Omron CX-Programmer project NewProject (CX-Programmer 9.80)

# PLC IN650_850: CJ2M CPU12
I/O table (CPU CJ2M-CPU12): rack 0 slot 1 CJ1W-ID211; rack 0 slot 2 CJ1W-ID211; rack 0 slot 3 CJ1W-OD212; rack 0 slot 4 CJ1W-OD212; rack 0 slot 5 CJ1W-OD212

## Global symbols (name address type ; comment)
ACC_Target_Frequency H31 DINT
ACC_accel_decel H30 UINT
AC_Drive_Fault W151.12 BOOL
AC_Drive_OK 1.07 BOOL  ; Drive OK output from infeed conveyor
ADV_ACC D882 DINT
ADV_ACC_4ms D1100 UINT
ADV_DEC D884 DINT
ADV_DEC_4ms D1104 UINT
ADV_Movement_Calcs Vel_ACC_DEC_Scale
ADV_Vel D886 DINT
Air_Pressure_Check T0160 TIMER  ; Debounce delay for Air Pressure
Air_Pressure_Fault W151.02 BOOL  ; Air Pressure Fault
Air_Pressure_OK 0.04 BOOL  ; Air Pressure switch
Analog_IO_Type D20001 CHANNEL  ; Analog input and output types.  Bit pattern of 1010101000000001 (#AA01) means all inputs are 4-20 mA and the output are 0 - 10VDC).
Analog_IO_Use_Config D20000 CHANNEL  ; #71 means that Inputs 1, 2 and 3 are used (bits 4, 5 and 6 on makes up 7 HEX) and output 1 is used (bit 0 on makes up 1 HEX).
2008 CHANNEL  ; top Vac sensor
D10000 CHANNEL  ; Vacuum graph 1 starting word
D10001 CHANNEL  ; top Vac scaled output
D10022 CHANNEL  ; scaled_measured_height_forHMI
D2041 CHANNEL  ; Unscaled Point A in slope
D2042 CHANNEL  ; Scaled Point B in slope
D2043 CHANNEL  ; Unscaled Point B in slope
D920 CHANNEL  ; Present value 1
D921 CHANNEL  ; Loop 2 Present value
D922 CHANNEL  ; Loop 3 Present value
D925 CHANNEL  ; Setpoint 1
T0226 BOOL  ; Delay down for lowering
T1103 BOOL  ; idel film time out
W497.00 BOOL  ; Temp bit HMI
Average_tray_height D2036 UINT  ; Average height of trays
Average_trays Average
Beginning_of_Cycle W202.06 BOOL  ; Beginning of the cycle
Break_Recover_Timer T1102 TIMER  ; Printer Film Break Delay
Calc_TPM TPM_Calc
Clear_Film_parameter_changed D2204.02 BOOL  ; Clear film parameter has changed
Close_Tool_Latch W200.12 BOOL
Cool_Timer T0124 TIMER  ; Cool Timer
CtoF C_to_F
Current1 D3005 CHANNEL  ; Stroom solid state 1
Current2 D3006 CHANNEL  ; Stroom solid state 2
Current3 D3007 CHANNEL  ; Stroom solid state 3
Current4 D3008 CHANNEL  ; Stroom solid state 4
Dancing_Timer T0203 TIMER  ; Dancing Timer
Dancing_Tray_Stop_Bit W200.14 BOOL
Data_Recipe_0 E0 CHANNEL[250]  ; All of the data for Recipe 0
Data_Recipe_1 E250 CHANNEL[250]  ; All of the data for Recipe 1
Data_Recipe_10 E2500 CHANNEL[250]  ; All of the data for Recipe 10
Data_Recipe_11 E2750 CHANNEL[250]  ; All of the data for Recipe 11
Data_Recipe_12 E3000 CHANNEL[250]  ; All of the data for Recipe 12
Data_Recipe_13 E3250 CHANNEL[250]  ; All of the data for Recipe 13
Data_Recipe_14 E3500 CHANNEL[250]  ; All of the data for Recipe 14
Data_Recipe_15 E3750 CHANNEL[250]  ; All of the data for Recipe 15
Data_Recipe_16 E4000 CHANNEL[250]  ; All of the data for Recipe 16
Data_Recipe_17 E4250 CHANNEL[250]  ; All of the data for Recipe 17
Data_Recipe_18 E4500 CHANNEL[250]  ; All of the data for Recipe 18
Data_Recipe_19 E4750 CHANNEL[250]  ; All of the data for Recipe 19
Data_Recipe_2 E500 CHANNEL[250]  ; All of the data for Recipe 2
Data_Recipe_20 E5000 CHANNEL[250]  ; All of the data for Recipe 20
Data_Recipe_21 E5250 CHANNEL[250]  ; All of the data for Recipe 21
Data_Recipe_22 E5500 CHANNEL[250]  ; All of the data for Recipe 22
Data_Recipe_23 E5750 CHANNEL[250]  ; All of the data for Recipe 23
Data_Recipe_24 E6000 CHANNEL[250]  ; All of the data for Recipe 24
Data_Recipe_25 E6250 CHANNEL[250]  ; All of the data for Recipe 25
Data_Recipe_26 E6500 CHANNEL[250]  ; All of the data for Recipe 26
Data_Recipe_27 E6750 CHANNEL[250]  ; All of the data for Recipe 27
Data_Recipe_28 E7000 CHANNEL[250]  ; All of the data for Recipe 28
Data_Recipe_29 E7250 CHANNEL[250]  ; All of the data for Recipe 29
Data_Recipe_3 E750 CHANNEL[250]  ; All of the data for Recipe 3
Data_Recipe_30 E7500 CHANNEL[250]  ; All of the data for Recipe 30
Data_Recipe_31 E7750 CHANNEL[250]  ; All of the data for Recipe 31
Data_Recipe_32 E8000 CHANNEL[250]  ; All of the data for Recipe 32
Data_Recipe_33 E8250 CHANNEL[250]  ; All of the data for Recipe 33
Data_Recipe_34 E8500 CHANNEL[250]  ; All of the data for Recipe 34
Data_Recipe_35 E8750 CHANNEL[250]  ; All of the data for Recipe 35
Data_Recipe_36 E9000 CHANNEL[250]  ; All of the data for Recipe 36
Data_Recipe_37 E9250 CHANNEL[250]  ; All of the data for Recipe 37
Data_Recipe_38 E9500 CHANNEL[250]  ; All of the data for Recipe 38
Data_Recipe_39 E9750 CHANNEL[250]  ; All of the data for Recipe 39
Data_Recipe_4 E1000 CHANNEL[250]  ; All of the data for Recipe 4
Data_Recipe_40 E10000 CHANNEL[250]  ; All of the data for Recipe 40
Data_Recipe_41 E10250 CHANNEL[250]  ; All of the data for Recipe 41
Data_Recipe_42 E10500 CHANNEL[250]  ; All of the data for Recipe 42
Data_Recipe_43 E10750 CHANNEL[250]  ; All of the data for Recipe 43
Data_Recipe_44 E11000 CHANNEL[250]  ; All of the data for Recipe 44
Data_Recipe_45 E11250 CHANNEL[250]  ; All of the data for Recipe 45
Data_Recipe_46 E11500 CHANNEL[250]  ; All of the data for Recipe 46
Data_Recipe_47 E11750 CHANNEL[250]  ; All of the data for Recipe 47
Data_Recipe_48 E12000 CHANNEL[250]  ; All of the data for Recipe 48
Data_Recipe_49 E12250 CHANNEL[250]  ; All of the data for Recipe 49
Data_Recipe_5 E1250 CHANNEL[250]  ; All of the data for Recipe 5
Data_Recipe_50 E12500 CHANNEL[250]  ; All of the data for Recipe 50
Data_Recipe_51 E12750 CHANNEL[250]  ; All of the data for Recipe 51
Data_Recipe_52 E13000 CHANNEL[250]  ; All of the data for Recipe 52
Data_Recipe_53 E13250 CHANNEL[250]  ; All of the data for Recipe 53
Data_Recipe_54 E13500 CHANNEL[250]  ; All of the data for Recipe 54
Data_Recipe_55 E13750 CHANNEL[250]  ; All of the data for Recipe 55
Data_Recipe_56 E14000 CHANNEL[250]  ; All of the data for Recipe 56
Data_Recipe_57 E14250 CHANNEL[250]  ; All of the data for Recipe 57
Data_Recipe_58 E14500 CHANNEL[250]  ; All of the data for Recipe 58
Data_Recipe_59 E14750 CHANNEL[250]  ; All of the data for Recipe 59
Data_Recipe_6 E1500 CHANNEL[250]  ; All of the data for Recipe 6
Data_Recipe_60 E15000 CHANNEL[250]  ; All of the data for Recipe 60
Data_Recipe_61 E15250 CHANNEL[250]  ; All of the data for Recipe 61
Data_Recipe_62 E15500 CHANNEL[250]  ; All of the data for Recipe 62
Data_Recipe_63 E15750 CHANNEL[250]  ; All of the data for Recipe 63
Data_Recipe_64 E16000 CHANNEL[250]  ; All of the data for Recipe 64
Data_Recipe_65 E16250 CHANNEL[250]  ; All of the data for Recipe 65
Data_Recipe_66 E16500 CHANNEL[250]  ; All of the data for Recipe 66
Data_Recipe_67 E16750 CHANNEL[250]  ; All of the data for Recipe 67
Data_Recipe_68 E17000 CHANNEL[250]  ; All of the data for Recipe 68
Data_Recipe_69 E17250 CHANNEL[250]  ; All of the data for Recipe 69
Data_Recipe_7 E1750 CHANNEL[250]  ; All of the data for Recipe 7
Data_Recipe_70 E17500 CHANNEL[250]  ; All of the data for Recipe 70
Data_Recipe_71 E17750 CHANNEL[250]  ; All of the data for Recipe 71
Data_Recipe_72 E18000 CHANNEL[250]  ; All of the data for Recipe 72
Data_Recipe_73 E18250 CHANNEL[250]  ; All of the data for Recipe 73
Data_Recipe_74 E18500 CHANNEL[250]  ; All of the data for Recipe 74
Data_Recipe_75 E18750 CHANNEL[250]  ; All of the data for Recipe 75
Data_Recipe_76 E19000 CHANNEL[250]  ; All of the data for Recipe 76
Data_Recipe_77 E19250 CHANNEL[250]  ; All of the data for Recipe 77
Data_Recipe_78 E19500 CHANNEL[250]  ; All of the data for Recipe 78
Data_Recipe_79 E19750 CHANNEL[250]  ; All of the data for Recipe 79
Data_Recipe_8 E2000 CHANNEL[250]  ; All of the data for Recipe 8
Data_Recipe_80 E20000 CHANNEL[250]  ; All of the data for Recipe 80
Data_Recipe_81 E20250 CHANNEL[250]  ; All of the data for Recipe 81
Data_Recipe_82 E20500 CHANNEL[250]  ; All of the data for Recipe 82
Data_Recipe_83 E20750 CHANNEL[250]  ; All of the data for Recipe 83
Data_Recipe_84 E21000 CHANNEL[250]  ; All of the data for Recipe 84
Data_Recipe_85 E21250 CHANNEL[250]  ; All of the data for Recipe 85
Data_Recipe_86 E21500 CHANNEL[250]  ; All of the data for Recipe 86
Data_Recipe_87 E21750 CHANNEL[250]  ; All of the data for Recipe 87
Data_Recipe_88 E22000 CHANNEL[250]  ; All of the data for Recipe 88
Data_Recipe_89 E22250 CHANNEL[250]  ; All of the data for Recipe 89
Data_Recipe_9 E2250 CHANNEL[250]  ; All of the data for Recipe 9
Data_Recipe_90 E22500 CHANNEL[250]  ; All of the data for Recipe 90
Data_Recipe_91 E22750 CHANNEL[250]  ; All of the data for Recipe 91
Data_Recipe_92 E23000 CHANNEL[250]  ; All of the data for Recipe 92
Data_Recipe_93 E23250 CHANNEL[250]  ; All of the data for Recipe 93
Data_Recipe_94 E23500 CHANNEL[250]  ; All of the data for Recipe 94
Data_Recipe_95 E23750 CHANNEL[250]  ; All of the data for Recipe 95
Data_Recipe_96 E24000 CHANNEL[250]  ; All of the data for Recipe 96
Data_Recipe_97 E24250 CHANNEL[250]  ; All of the data for Recipe 97
Data_Recipe_98 E24500 CHANNEL[250]  ; All of the data for Recipe 98
Data_Recipe_99 E24750 CHANNEL[250]  ; All of the data for Recipe 99
Debounce_TS1 T0100 TIMER  ; Debounce timer for sensor at Tray Stop 1
Debounce_TS2 T0101 TIMER  ; Debounce timer for sensor at Tray Stop 2
Debounce_TS3 T0102 TIMER  ; Debounce timer for sensor at Tray Stop 3
Debounce_TS4 T0103 TIMER  ; Debounce timer for sensor at Tray Stop 4
Debounce_TS5 T0104 TIMER  ; Debounce timer for sensor at Tray Stop 5
Default_Recipe_Data E26000 CHANNEL[250]  ; Default recipe data used when erasing a recipe
Delay_on_upstream D280 UINT
Demo_Mode W200.10 BOOL  ; With or without trays
Demo_Mode_No_Trays W201.00 BOOL
Demo_Mode_With_Trays W201.01 BOOL
Disable_Gas_Delay W250.05 BOOL  ; Disables Input on the HMI
Disable_Gas_Duration W250.06 BOOL  ; Disables Input on the HMI
Disable_Gas_Pressure W250.07 BOOL  ; Disables Input on the HMI
Disable_Seal_Delay W250.10 BOOL  ; Disables Input on the HMI
Disable_Seal_Duration W250.11 BOOL  ; Disables Input on the HMI
Disable_Stepper_out 2961.04 BOOL
Disable_Tool_Open_Delay W250.12 BOOL  ; Disables Input on the HMI
Disable_Vac_Bottom_Delay W250.01 BOOL  ; Disables Input on the HMI
Disable_Vac_Extra W250.04 BOOL  ; Disables Input on the HMI
Disable_Vac_Top_Delay W250.00 BOOL  ; Disables Input on the HMI
Disable_Vac_duration W250.02 BOOL  ; Disables Input on the HMI
Disable_Vac_pressure W250.03 BOOL  ; Disables Input on the HMI
Disable_Vent_Pressure W250.09 BOOL  ; Disables Input on the HMI
Disable_Vent_Top_Delay W250.08 BOOL  ; Disables Input on the HMI
Disable_by_Pressure W202.08 BOOL  ; Disable vac, gas and vent by pressure buttons
Door_Open_Fault W151.01 BOOL  ; Door open
DownStream_Alarm W154.00 BOOL  ; Downstream alarm message bit
Downstream_bypass D2009.13 BOOL  ; Bypass Downstream input
Enable_Analog_Out 2000.00 BOOL  ; enables analog output for speed reference to AC Drive.
Execute_slow_down D2204.01 BOOL
Eye_mark_selection D2300.00 BOOL  ; Single Eye Mark per move selected
FILMREG_ESTOP_DECEL H50 UINT  ; H50 Film Reg E-Stop Decel
FILMREG_ESTOP_FREQ H51 DINT  ; H51/H52 Film Reg E-Stop Target Freq
FILM_DIST_REVYANK_REGIST D1158 DINT
Fault_Exists W156.15 BOOL  ; A fault exists
File_Mem_Operation_Flag A343.13 BOOL  ; File memory operation in progress.
File_Write_Read_Destination D1450 WORD[4]  ; Destination word for FWRIT and FREAD instructions
FilmReg_Started W203.15 BOOL  ; Film Feed with Registration Started
FilmScaling Film_Scaling
Film_Accel_Rate H0 UINT
Film_Advance_button_timer T0125 TIMER  ; Timer for Film Advance button
Film_Decel_Rate H1 UINT
Film_No_Origin_Flag A280.05 BOOL  ; No Origin Established
Film_Present_Position A276 DINT  ; Current position of the film axis
Film_Pulse_Error_Flag A280.07 BOOL  ; Pulse output error
Film_Pulse_Out_Complete A280.03 BOOL  ; Pulse Output complete
Film_Pulse_interrupt_Feed_Flag A280.08 BOOL  ; Interrupt feeding (Registration) is in progress.
Film_Pulses_Ongoing A280.04 BOOL  ; Film feeding is in process
Film_Pulses_Output_Status A280.00 BOOL  ; OFF - Constant speed, ON - Accelerating / decelerating
Film_Reg_Fault_Delay T0152 TIMER
Film_Reg_check_Failed W204.00 BOOL  ; Check at end of film reg feed for problems
Film_Registration_Distance_Calc D1120 DINT
Film_Slow_Down_Speed D246 UINT  ; Slow Down Speed for Registration
Film_Starting_Freq H6 DINT
Film_Target_Frequency H2 DINT
Film_Target_Position H4 DINT
FlSaveLoop1 W502.00 BOOL  ; FlSaveLoop1
FlSaveLoop2 W502.01 BOOL  ; FlSaveLoop2
FlSaveLoop3 W502.02 BOOL  ; FlSaveLoop3
FlSaveLoop4 W502.03 BOOL  ; FlSaveLoop4
FlSaveLoop5 W502.04 BOOL  ; FlSaveLoop5
FlSaveLoop6 W502.05 BOOL  ; FlSaveLoop6
Flat_Pack_Mode W201.02 BOOL
Forced_Bit_Status_Fault W151.03 BOOL  ; There is a bit forced.
Front_Gripper_Closed_Prox 0.07 BOOL  ; Front Gripper closed proximity sw
Front_Gripper_Open_Prox 0.06 BOOL  ; Front Gripper open proximity switch
FtoC F_to_C
Gas_Delay_Simultaneous_Timer T0206 TIMER  ; Used for simultaneous Mode
Gas_Delay_Timer T0117 TIMER  ; Gas Delay Timer
Gas_Duration_Simultaneous_Timer T0205 TIMER  ; Used for simultaneous Mode
Gas_Duration_Timer T0118 TIMER  ; Gas Duration Timer
Gas_Pressure_Check T0161 TIMER  ; Debounce delay for Gas Pressure
Gas_Pressure_Fault_Timer T0221 TIMER  ; Allows for dip in pressure during map cycle
Gas_Pressure_Low_Fault W151.13 BOOL  ; Gas Pressure low
Gas_Pressure_OK 0.05 BOOL  ; Gas Pressure Switch
Gas_Pulse 2011.03 BOOL  ; gas_pulse_latch
Gas_Timeout_WD_Fault W150.04 BOOL  ; Watchdog Timer Fault
Gas_Timeout_WD_Timer T0133 TIMER  ; Watchdog Timer
Gas_level_chosen D2035 UINT  ; Gas level used on next tool cycle
Gas_level_used_in_cycle D2039 UINT  ; Value used for next cycle
Gas_range_scale D2040 LWORD  ; Scaled Point A in slope
Gate_Sensor1_Filter T0243 TIMER  ; Gate Sensor 1 Filter
Gate_Sensor2_Filter T0244 TIMER  ; Gate Sensor 2 Filter
Gate_Sensor3_Filter T0245 TIMER  ; Gate Sensor 3 Filter
Gate_Sensor4_Filter T0246 TIMER  ; Gate Sensor 4 Filter
Gate_Sensor5_Filter T0247 TIMER  ; Gate Sensor 5 Filter
GripperClose_DoubleHitPrevent W104.06 BOOL
GripperOpen_Time_doubleHitPrevent W104.05 BOOL
Gripper_ADV_Delay_Timer T0107 TIMER  ; Gripper Advance delay
Gripper_ADV_WD_Fault W150.02 BOOL  ; Watchdog Timer Fault
Gripper_ADV_WD_Timer T0131 TIMER  ; Watchdog Timer
Gripper_Accel_Rate H10 UINT
Gripper_Advance_Command W200.02 BOOL  ; Gripper Advance command
Gripper_Advance_Complete W200.09 BOOL  ; Gripper has advanced
Gripper_Close_Delay_Timer T0105 TIMER  ; Gripper Close Delay
Gripper_Close_Delay_Timer_Jog T0501 TIMER  ; Delays jog to charge cylinder
Gripper_Close_WD_Fault W150.00 BOOL  ; Watchdog Timer Fault
Gripper_Close_WD_Timer T0129 TIMER  ; Watchdog Timer
Gripper_Decel_Rate H11 UINT
Gripper_Extended_Prox 0.08 BOOL  ; Gripper extended proximity sw
Gripper_Homed W200.01 BOOL  ; Gripper has been homed
Gripper_No_Origin_Flag A281.05 BOOL  ; No Origin Established
Gripper_Open_Delay_timer T0106 TIMER  ; Gripper Open delay
Gripper_Open_WD_Fault W150.01 BOOL  ; Watchdog Timer Fault
Gripper_Open_WD_Timer T0130 TIMER  ; Watchdog Timer
Gripper_Present_Position A278 DINT  ; Current position of the gripper axis
Gripper_Pulse_Error_Flag A281.07 BOOL  ; Pulse output error
Gripper_Pulse_Interrupt_Feed_Flag A281.08 BOOL  ; Interrupt feeding (Registration) is in progress.
Gripper_Pulse_Out_Complete A281.03 BOOL  ; Pulse Output complete
Gripper_Pulses_Output_Status A281.00 BOOL  ; OFF - Constant speed, ON - Accelerating / decelerating
Gripper_RET_WD_Fault W150.03 BOOL  ; Watchdog Timer Fault
Gripper_RET_WD_Timer T0132 TIMER  ; Watchdog Timer
Gripper_Retract_Command W200.03 BOOL  ; Gripper Retract command
Gripper_Retract_Complete W200.08 BOOL  ; Gripper has retracted
Gripper_Retract_Delay T0229 TIMER  ; Delay to keep IN450 Gripper Extend ON briefly
Gripper_Retracted_Prox 0.09 BOOL  ; Gripper retracted proximity sw
Gripper_Seq_Step_Number D510 UINT  ; Contains the step number for the gripper sequence
Gripper_Starting_Freq H16 DINT
Gripper_Target_Frequency H12 DINT
Gripper_Target_Position H14 DINT
Grippers_Closed W203.03 BOOL  ; Overall closed status
Grippers_Open W203.02 BOOL  ; Overall open status
Guard_Authority 0.15 BOOL  ; Safety controller Input
Guard_OK 0.11 BOOL  ; Guard door switches ok
Guard_door_input 1.11 BOOL  ; Guard door input from safety switch (SI6)
HMI_Change_Screen_Number D901 UINT  ; Change this register to change screens
HMI_Clean_Infeed_Speed D874 UINT
HMI_Cleaning_Tool_Sealed W102.03 BOOL
HMI_Close_Tool_Cleaning W102.00 BOOL
HMI_Copy_Recipe W103.13 BOOL
HMI_Copy_Recipe_Number D875 UINT
HMI_Current_Screen D900 UINT  ; Screen number of current screen
HMI_Day D835 UINT  ; Day
HMI_Delete_Recipe W103.11 BOOL
HMI_Disengage_Tool_Disable W101.14 BOOL
HMI_Display_Pressure_mbar D806 UINT  ; Pressure
HMI_Engage_Tool_Disable W101.15 BOOL
HMI_Export_All_recipe W103.14 BOOL
HMI_Film_ADV_Command W100.12 BOOL
HMI_Film_ADV_State D855 UINT
HMI_Film_ADV_Time D844 UINT
HMI_Film_ADV_Time_Bit W201.10 BOOL  ; Allows time to be calculated
HMI_Film_ADV_Time_Temp D1126 UINT  ; Temporary register for time value
HMI_Film_PB W100.05 BOOL  ; Film PB on HMI
HMI_Gas_Command W101.02 BOOL
HMI_Gas_Light W102.10 BOOL
HMI_Gas_State D861 UINT
HMI_Gas_Time D843 UINT
HMI_Gas_Time_Bit W201.09 BOOL  ; Allows time to be calculated
HMI_Gas_Time_Temp D1125 UINT  ; Temporary register for time value
HMI_Gas_Timeout D823 UINT  ; Gas Timeout
HMI_Grip_ADV_Command W100.15 BOOL
HMI_Grip_ADV_State D858 UINT
HMI_Grip_ADV_Time D850 UINT
HMI_Grip_ADV_Time_Bit W202.00 BOOL  ; Allows time to be calculated
HMI_Grip_ADV_Time_Temp D1132 UINT  ; Temporary register for time value
HMI_Grip_Close_Command W100.13 BOOL
HMI_Grip_Close_State D856 UINT
HMI_Grip_Close_Time D849 UINT
HMI_Grip_Close_Time_Bit W201.15 BOOL  ; Allows time to be calculated
HMI_Grip_Close_Time_Temp D1131 UINT  ; Temporary register for time value
HMI_Grip_Open_Command W100.14 BOOL
HMI_Grip_Open_State D857 UINT
HMI_Grip_Open_Time D848 UINT
HMI_Grip_Open_Time_Bit W201.14 BOOL  ; Allows time to be calculated
HMI_Grip_Open_Time_Temp D1130 UINT  ; Temporary register for time value
HMI_Grip_RET_Command W101.00 BOOL
HMI_Grip_RET_State D859 UINT
HMI_Grip_RET_Time D851 UINT
HMI_Grip_RET_Time_Bit W202.01 BOOL  ; Allows time to be calculated
HMI_Grip_RET_Time_Temp D1133 UINT  ; Temporary register for time value
HMI_Gripper_Adv_Time D821 UINT  ; Gripper Advance Time
HMI_Gripper_Close_Time D819 UINT  ; Gripper close Time
HMI_Gripper_Current_Pos D810 UINT  ; Current Position of Gripper
HMI_Gripper_Encoder_Scale D815 UINT  ; Gripper Encoder Scale
HMI_Gripper_Home_Speed D811 UINT  ; Gripper Home speed
HMI_Gripper_Jog_Accel D813 UINT  ; Gripper Jog Accel
HMI_Gripper_Jog_Decel D814 UINT  ; Gripper Jog Decel
HMI_Gripper_Jog_Velocity D812 UINT  ; Gripper Jog Velocity
HMI_Gripper_Max_Accel D817 UINT  ; Gripper Max Accel
HMI_Gripper_Max_Velocity D816 UINT  ; Gripper Max Velocity
HMI_Gripper_Open_Time D820 UINT  ; Gripper Open Time
HMI_Gripper_Pos_Tolerance D818 UINT  ; Gripper Position Tolerance
HMI_Gripper_Ret_Time D822 UINT  ; Gripper Return Time
HMI_Guard_Warning W100.03 BOOL  ; The guard is open
HMI_Heat_PM W100.07 BOOL  ; Heat PB on HMI
HMI_High_Tolerance D933 UINT
HMI_Hour D837 UINT  ; Hour
HMI_Import_All_Recipe W103.15 BOOL
HMI_Jog_PB W100.04 BOOL  ; Jog PB on HMI
HMI_Leak_By_Pressure W101.10 BOOL
HMI_Leak_Pressure D873 UINT
HMI_Leak_Rate_Display D871 UINT
HMI_Leak_Time_Display D870 UINT
HMI_Lift_Down_Time D828 UINT  ; Lift down time
HMI_Lift_Up_Time D827 UINT  ; Lift Up time
HMI_Live_Pressure_Display D867 UINT
HMI_Load_Recipe W103.08 BOOL
HMI_Lock_Tool W101.13 BOOL  ; HMI - Lock Upper Tool
HMI_Low_Tolerance D931 UINT
HMI_Lower_Vac_Command W101.05 BOOL
HMI_Lower_Vac_Light W102.09 BOOL
HMI_Lower_Vac_State D864 UINT
HMI_Lower_Vent_Command W101.07 BOOL
HMI_Lower_Vent_Light W102.12 BOOL
HMI_Lower_Vent_State D866 UINT
HMI_MAP_Cycle_Command W101.01 BOOL
HMI_MAP_Cycle_State D860 UINT
HMI_Machine_Config D1143 UINT
HMI_Map_Cycle_Time D845 UINT
HMI_Map_Cycle_Time_Bit W201.11 BOOL  ; Allows time to be calculated
HMI_Map_Cycle_Time_Temp D1127 UINT  ; Temporary register for time value
HMI_Max_SP D927 UINT
HMI_Max_Set_Temp D831 UINT  ; Max Temperature
HMI_Max_Temp_Allowed D1135 INT  ; Maximum allowed setting for HMI
HMI_Min D838 UINT  ; Minutes
HMI_Min_Temp_allowed D1134 INT  ; Minimum allowed setting for HMI
HMI_Month D834 UINT  ; Month
HMI_Open_Cleaning W102.02 BOOL
HMI_Open_Gripper_Auto D2011.01 BOOL  ; Enable Gripper Open on Reset
HMI_Operator_Gas W104.02 BOOL
HMI_Overtemp D832 INT  ; Overtemp
HMI_Overtemp_SP D929 UINT
HMI_PID_Mode W501.09 BOOL  ; HMI PID Mode Select-Default/Custom
HMI_Pump_PB W100.06 BOOL  ; Pump PB on HMI
HMI_Recipe_Selection_0 W102.14 BOOL
HMI_Recipe_Selection_1 W102.15 BOOL
HMI_Recipe_Selection_2 W103.00 BOOL
HMI_Recipe_Selection_3 W103.01 BOOL
HMI_Recipe_Selection_4 W103.02 BOOL
HMI_Recipe_Selection_5 W103.03 BOOL
HMI_Recipe_Selection_6 W103.04 BOOL
HMI_Recipe_Selection_7 W103.05 BOOL
HMI_Recipe_Selection_8 W103.06 BOOL
HMI_Recipe_Selection_9 W103.07 BOOL
HMI_Recipe_has_Changed W100.08 BOOL  ; Recipe has changed indicator
HMI_Rename_Recipe W103.12 BOOL
HMI_Reset_Counter W104.01 BOOL  ; HMI Reset Count PB
HMI_Reset_PB W100.02 BOOL  ; Reset PB on HMI
HMI_Result_Time_Display D869 UINT
HMI_Rewind_Timeout D830 UINT  ; Rewind Timeout
HMI_Run_Infeed_Cleaning W102.01 BOOL
HMI_Run_Outfeed_Conveyor W104.03 BOOL  ; Run Outfeed from HMI
HMI_Run_Vacuum_Pump W101.11 BOOL
HMI_Run_Vacuum_Test W101.08 BOOL
HMI_Save_As_Name D1000 STRING[38]  ; Save as name
HMI_Save_Loaded_Recipe W103.09 BOOL
HMI_Save_Recipe_As W103.10 BOOL
HMI_SealPause_PB W503.05 BOOL  ; Seal Pause PB HMI on
HMI_Seal_Command W101.03 BOOL
HMI_Seal_Light W102.13 BOOL
HMI_Seal_State D862 UINT
HMI_Sec D839 UINT  ; Seconds
HMI_Select_Recipe W104.00 BOOL
HMI_Servo_End_of_Stroke_Max D1145 UINT
HMI_Servo_End_of_Stroke_Min D1144 UINT
HMI_Sleep_Mode_Enable W202.09 BOOL  ; On = Sleep mode enabled Off = Sleep Mode Disabled
HMI_Sleep_Mode_Temp D935 UINT
HMI_Star_Pressure_Display D868 UINT
HMI_Start_PB W100.00 BOOL  ; Green Start PB
HMI_Stop_PB W100.01 BOOL  ; Red Stop PB
HMI_Target_Pressure D872 UINT
HMI_Temp_Display1 D920 UINT  ; Temp Display 1
HMI_Temp_Display2 D921 UINT  ; Temp Display 2
HMI_Temp_Display3 D922 UINT  ; Temp Display 3
HMI_Temp_Display4 D923 UINT  ; Temp Display 4
HMI_Temp_Display5 D924 UINT  ; Temp Display 5
HMI_Temp_High_Tolerance D894 INT  ; Temperature Tolerance - Max side
HMI_Temp_Low_Tolerance D833 INT  ; Temperature Tolerance - Min side
HMI_Temp_Setpoint D925 UINT
HMI_Tool_Change_Position D1146 DINT  ; Tool Change Position
HMI_Tool_Down_Command W100.11 BOOL
HMI_Tool_Down_State D854 UINT
HMI_Tool_Down_Time D847 UINT
HMI_Tool_Down_Time_Bit W201.13 BOOL  ; Allows time to be calculated
HMI_Tool_Down_Time_Temp D1129 UINT  ; Temporary register for time value
HMI_Tool_Light W102.07 BOOL
HMI_Tool_Unlock_Command W100.09 BOOL
HMI_Tool_Unlock_State D852 UINT
HMI_Tool_Up_Command W100.10 BOOL
HMI_Tool_Up_State D853 UINT
HMI_Tool_Up_Time D846 UINT
HMI_Tool_Up_Time_Bit W201.12 BOOL  ; Allows time to be calculated
HMI_Tool_Up_Time_Temp D1128 UINT  ; Temporary register for time value
HMI_Total_Cycle_Time D840 UINT
HMI_Total_Cycle_Time_Bit W201.06 BOOL  ; Allows time to be calculated
HMI_Total_Cycle_Time_Temp D1122 UINT  ; Temporary register for time value
HMI_Tray_Delay_Time D841 UINT
HMI_Tray_Delay_Time_Bit W201.07 BOOL  ; Allows time to be calculated
HMI_Tray_Delay_Time_Temp D1123 UINT  ; Temporary register for time value
HMI_Unlock_Tool W101.12 BOOL  ; HMI - Unlock Upper Tool
HMI_Upper_Tool_Lock_Time D825 UINT  ; Upper Tool Lock Time
HMI_Upper_Tool_Unlock_Time D826 UINT  ; Upper tool unlock time
HMI_Upper_Vac_Command W101.04 BOOL
HMI_Upper_Vac_Light W102.08 BOOL
HMI_Upper_Vac_State D863 UINT
HMI_Upper_Vent_Command W101.06 BOOL
HMI_Upper_Vent_Light W102.11 BOOL
HMI_Upper_Vent_State D865 UINT
HMI_Use_Printer D28.15 BOOL  ; Use printer selection on Machine Config Screen
HMI_Vac_Time D842 UINT
HMI_Vac_Time_Bit W201.08 BOOL  ; Allows time to be calculated
HMI_Vac_Time_Temp D1124 UINT  ; Temporary register for time value
HMI_Vac_Timeout D824 UINT  ; Vac Timeout
HMI_Vacuum_By_Pressure W101.09 BOOL
HMI_Vent_Timeout D829 UINT  ; Vent Timeout
HMI_Year D836 UINT  ; Year
High_Temp_Tol_CtoF offsetC_to_offsetF
High_Temp_Tol_FtoC OffsetF_to_OffsetC
IN450_Machine W203.00 BOOL  ; The machine is either an IN450 or IN450 Plus
IN450_Mode W202.10 BOOL
IN450_Plus_Mode W202.11 BOOL
IN650_850_Machine W203.01 BOOL  ; The machine is either an IN650 or IN850
IN650_Mode W202.12 BOOL
IN850_Mode W202.13 BOOL
Idle_Film_Feed W104.04 BOOL
Idle_Film_Feed_Running W300.00 BOOL
Idle_Film_SP_secs D964 UDINT  ; Idle time Setpoint in 0.1s units
Idle_Film_Timer T0223 TIMER
Idle_Film_time_SP D963 UINT  ; Time to wait to advance film after sitting idle in minutes
Idle_Film_timer_Seconds D2203 UINT
Ignore_eye_marks D2300.01 BOOL
Infeed_Conveyor_Run 3.07 BOOL  ; Run to A4 Infeed conveyor VFD
Infeed_Conveyor_speed_ref 2001 UINT  ; Analog output for speed reference to AC Drive 0 - 7999 = 0 - 10VDC
Infeed_Conveyor_speed_register D1116 UINT  ; Register for the speed reference.  It gets it from D34 or D874 for normal operation or Clean Mode
Infeed_Debounce_Timer T0108 TIMER  ; Infeed debounce timer
Infeed_Estop_Fault W150.15 BOOL  ; Infeed E-stop pressed
Infeed_Estop_OK 0.01 BOOL  ; E-Stop circuit status
Infeed_Gate_Down_Delay T0204 TIMER
Infeed_Gate_Sensor 0.12 BOOL  ; Infeed Gate Sensor
Infeed_Gate_Seq_Step_Number D509 UINT  ; Contains the step number for the infeed gate sequence
Infeed_Sensor_Off_Filter_Timer T0261 TIMER
Infeed_Sensor_On_Filter_Timer T0260 TIMER
Infeed_Seq_Step_Number D508 UINT  ; Contains the step number for the Infeed sequence
Infeed_Stop_Delay T0109 TIMER  ; Infeed stop delay
Infeed_Stop_Retry_Delay T0111 TIMER  ; Retry timer to send in a tray after missed tray
Infeed_Tray_Measure_Alarm W151.14 BOOL  ; Photo measurement of tray alarm
Infeed_stop_delay_bit W200.15 BOOL
Initialize_Bar D802 UINT  ; Initialization status bar on HMI
Internal_Grip_ADV_State D958 UINT
Internal_Grip_Close_State D956 UINT
Internal_Grip_Open_State D957 UINT
Internal_Grip_RET_State D959 UINT
Internal_Tool_Down_State D954 UINT
Internal_Tool_Up_State D953 UINT
Jog_Scaling Film_Scaling
Jog_Target_Frequency H33 DINT
Jog_accel_decel H32 UINT
K1_Remote_Stop_IN 0.13 BOOL  ; K1 Remote Stop FROM Plant equipment input
K2_Vacuum_Pump_Run 2.05 BOOL  ; K2 Vacuum Pump Run output
K3_Remote_Stop_OUT 3.10 BOOL  ; K3 Remote Stop TO Plant Equip.
Keyswitch_input_High_ox 1.13 BOOL  ; Keyswitch input to enable highox (simultaneous)
Last_High_Tolerance D934 UINT
Last_Loaded_Recipe_Advance_Accel D3071 UINT
Last_Loaded_Recipe_Advance_Decel D3072 UINT
Last_Loaded_Recipe_Advance_Time D3069 UINT
Last_Loaded_Recipe_Advance_Velocity D3070 UINT
Last_Loaded_Recipe_Bottom_Vacuum_Delay D3036 UINT
Last_Loaded_Recipe_Cycle_Type D3029 UINT  ; Cycle type selection (Flat, Map, Simultaneous, VSP)
Last_Loaded_Recipe_Dancing_Stop D3058 UINT
Last_Loaded_Recipe_Feed_Delay_After_Adv D3052 UINT
Last_Loaded_Recipe_Film_Feed_Accel D3076 UINT
Last_Loaded_Recipe_Film_Feed_Decel D3077 UINT
Last_Loaded_Recipe_Film_Feed_Velocity D3075 UINT
Last_Loaded_Recipe_Film_Jog_Accel D3080 UINT
Last_Loaded_Recipe_Film_Jog_Decel D3081 UINT
Last_Loaded_Recipe_Film_Jog_Velocity D3079 UINT
Last_Loaded_Recipe_Film_Length D3031 UINT  ; Film length to feed
Last_Loaded_Recipe_Gas_Delay D3040 UINT
Last_Loaded_Recipe_Gas_Duration D3041 UINT
Last_Loaded_Recipe_Gas_Pressure_SP D3042 UINT
Last_Loaded_Recipe_Gas_Type D3020.01 BOOL  ; Gas type - ON = Pressure, OFF = Time
Last_Loaded_Recipe_Grip_Open_Delay D3067 UINT
Last_Loaded_Recipe_Gripper_ADV_Delay D3057 UINT
Last_Loaded_Recipe_Gripper_Close_Delay D3050 UINT
Last_Loaded_Recipe_Infeed_Gate_Eye_Debounce D3055 UINT
Last_Loaded_Recipe_Infeed_speed D3034 UINT  ; Infeed speed setting
Last_Loaded_Recipe_Lift_Decel D3073 UINT
Last_Loaded_Recipe_Lost_Tray_Reset_Delay D3054 UINT
Last_Loaded_Recipe_Lower_Decel D3074 UINT
Last_Loaded_Recipe_Motion_Setting_from_Time D3020.05 BOOL  ; Chooses time setting or vel, accel and decel settings
Last_Loaded_Recipe_Name D3000 STRING[38]  ; Job name for Recipe 0 - 38 characters
Last_Loaded_Recipe_Number D3019 CHANNEL  ; Recipe Number (0 - 99)
Last_Loaded_Recipe_Number_of_Trays D3059 UINT
Last_Loaded_Recipe_REV_Yank D3020.03 BOOL  ; On if reverse yank enabled for film
Last_Loaded_Recipe_Reg_Offset D3033 UINT  ; Registration Offset
Last_Loaded_Recipe_Reg_enable D3020.04 BOOL  ; On if registration enabled for film
Last_Loaded_Recipe_Return_Accel D3065 UINT
Last_Loaded_Recipe_Return_Decel D3066 UINT
Last_Loaded_Recipe_Return_Time D3063 UINT
Last_Loaded_Recipe_Return_Velocity D3064 UINT
Last_Loaded_Recipe_Rev_Yank_Dist D3032 UINT  ; Reverse Yank Distance
Last_Loaded_Recipe_Rewind_On_Delay D3051 UINT
Last_Loaded_Recipe_Seal_Cool D3049 UINT
Last_Loaded_Recipe_Seal_Delay D3047 UINT
Last_Loaded_Recipe_Seal_Duration D3048 UINT
Last_Loaded_Recipe_Spare_Bits_WD0_bit10 D3020.10 BOOL  ; Spare
Last_Loaded_Recipe_Spare_Bits_WD0_bit11 D3020.11 BOOL  ; Spare
Last_Loaded_Recipe_Spare_Bits_WD0_bit12 D3020.12 BOOL  ; Spare
Last_Loaded_Recipe_Spare_Bits_WD0_bit13 D3020.13 BOOL  ; Spare
Last_Loaded_Recipe_Spare_Bits_WD0_bit14 D3020.14 BOOL  ; Spare
Last_Loaded_Recipe_Spare_Bits_WD0_bit15 D3020.15 BOOL  ; Spare
Last_Loaded_Recipe_Spare_Bits_WD0_bit6 D3020.06 BOOL  ; Spare
Last_Loaded_Recipe_Spare_Bits_WD0_bit7 D3020.07 BOOL  ; Spare
Last_Loaded_Recipe_Spare_Bits_WD0_bit8 D3020.08 BOOL  ; Spare
Last_Loaded_Recipe_Spare_Bits_WD0_bit9 D3020.09 BOOL  ; Spare
Last_Loaded_Recipe_Spare_Bits_WD1_bit0 D3021.00 BOOL  ; Spare
Last_Loaded_Recipe_Spare_Bits_WD1_bit1 D3021.01 BOOL  ; Spare
Last_Loaded_Recipe_Spare_Bits_WD1_bit10 D3021.10 BOOL  ; Spare
Last_Loaded_Recipe_Spare_Bits_WD1_bit11 D3021.11 BOOL  ; Spare
Last_Loaded_Recipe_Spare_Bits_WD1_bit12 D3021.12 BOOL  ; Spare
Last_Loaded_Recipe_Spare_Bits_WD1_bit13 D3021.13 BOOL  ; Spare
Last_Loaded_Recipe_Spare_Bits_WD1_bit14 D3021.14 BOOL  ; Spare
Last_Loaded_Recipe_Spare_Bits_WD1_bit15 D3021.15 BOOL  ; Spare
Last_Loaded_Recipe_Spare_Bits_WD1_bit2 D3021.02 BOOL  ; Spare
Last_Loaded_Recipe_Spare_Bits_WD1_bit3 D3021.03 BOOL  ; Spare
Last_Loaded_Recipe_Spare_Bits_WD1_bit4 D3021.04 BOOL  ; Spare
Last_Loaded_Recipe_Spare_Bits_WD1_bit5 D3021.05 BOOL  ; Spare
Last_Loaded_Recipe_Spare_Bits_WD1_bit6 D3021.06 BOOL  ; Spare
Last_Loaded_Recipe_Spare_Bits_WD1_bit7 D3021.07 BOOL  ; Spare
Last_Loaded_Recipe_Spare_Bits_WD1_bit8 D3021.08 BOOL  ; Spare
Last_Loaded_Recipe_Spare_Bits_WD1_bit9 D3021.09 BOOL  ; Spare
Last_Loaded_Recipe_Spare_Bits_WD2_bit0 D3022.00 BOOL  ; Spare
Last_Loaded_Recipe_Spare_Bits_WD2_bit1 D3022.01 BOOL  ; Spare
Last_Loaded_Recipe_Spare_Bits_WD2_bit10 D3022.10 BOOL  ; Spare
Last_Loaded_Recipe_Spare_Bits_WD2_bit11 D3022.11 BOOL  ; Spare
Last_Loaded_Recipe_Spare_Bits_WD2_bit12 D3022.12 BOOL  ; Spare
Last_Loaded_Recipe_Spare_Bits_WD2_bit13 D3022.13 BOOL  ; Spare
Last_Loaded_Recipe_Spare_Bits_WD2_bit14 D3022.14 BOOL  ; Spare
Last_Loaded_Recipe_Spare_Bits_WD2_bit15 D3022.15 BOOL  ; Spare
Last_Loaded_Recipe_Spare_Bits_WD2_bit2 D3022.02 BOOL  ; Spare
Last_Loaded_Recipe_Spare_Bits_WD2_bit3 D3022.03 BOOL  ; Spare
Last_Loaded_Recipe_Spare_Bits_WD2_bit4 D3022.04 BOOL  ; Spare
Last_Loaded_Recipe_Spare_Bits_WD2_bit5 D3022.05 BOOL  ; Spare
Last_Loaded_Recipe_Spare_Bits_WD2_bit6 D3022.06 BOOL  ; Spare
Last_Loaded_Recipe_Spare_Bits_WD2_bit7 D3022.07 BOOL  ; Spare
Last_Loaded_Recipe_Spare_Bits_WD2_bit8 D3022.08 BOOL  ; Spare
Last_Loaded_Recipe_Spare_Bits_WD2_bit9 D3022.09 BOOL  ; Spare
Last_Loaded_Recipe_Spare_Bits_WD3_bit0 D3023.00 BOOL  ; Spare
Last_Loaded_Recipe_Spare_Bits_WD3_bit1 D3023.01 BOOL  ; Spare
Last_Loaded_Recipe_Spare_Bits_WD3_bit10 D3023.10 BOOL  ; Spare
Last_Loaded_Recipe_Spare_Bits_WD3_bit11 D3023.11 BOOL  ; Spare
Last_Loaded_Recipe_Spare_Bits_WD3_bit12 D3023.12 BOOL  ; Spare
Last_Loaded_Recipe_Spare_Bits_WD3_bit13 D3023.13 BOOL  ; Spare
Last_Loaded_Recipe_Spare_Bits_WD3_bit14 D3023.14 BOOL  ; Spare
Last_Loaded_Recipe_Spare_Bits_WD3_bit15 D3023.15 BOOL  ; Spare
Last_Loaded_Recipe_Spare_Bits_WD3_bit2 D3023.02 BOOL  ; Spare
Last_Loaded_Recipe_Spare_Bits_WD3_bit3 D3023.03 BOOL  ; Spare
Last_Loaded_Recipe_Spare_Bits_WD3_bit4 D3023.04 BOOL  ; Spare
Last_Loaded_Recipe_Spare_Bits_WD3_bit5 D3023.05 BOOL  ; Spare
Last_Loaded_Recipe_Spare_Bits_WD3_bit6 D3023.06 BOOL  ; Spare
Last_Loaded_Recipe_Spare_Bits_WD3_bit7 D3023.07 BOOL  ; Spare
Last_Loaded_Recipe_Spare_Bits_WD3_bit8 D3023.08 BOOL  ; Spare
Last_Loaded_Recipe_Spare_Bits_WD3_bit9 D3023.09 BOOL  ; Spare
Last_Loaded_Recipe_Spare_Bits_WD4_bit0 D3024.00 BOOL  ; Spare
Last_Loaded_Recipe_Spare_Bits_WD4_bit1 D3024.01 BOOL  ; Spare
Last_Loaded_Recipe_Spare_Bits_WD4_bit10 D3024.10 BOOL  ; Spare
Last_Loaded_Recipe_Spare_Bits_WD4_bit11 D3024.11 BOOL  ; Spare
Last_Loaded_Recipe_Spare_Bits_WD4_bit12 D3024.12 BOOL  ; Spare
Last_Loaded_Recipe_Spare_Bits_WD4_bit13 D3024.13 BOOL  ; Spare
Last_Loaded_Recipe_Spare_Bits_WD4_bit14 D3024.14 BOOL  ; Spare
Last_Loaded_Recipe_Spare_Bits_WD4_bit15 D3024.15 BOOL  ; Spare
Last_Loaded_Recipe_Spare_Bits_WD4_bit2 D3024.02 BOOL  ; Spare
Last_Loaded_Recipe_Spare_Bits_WD4_bit3 D3024.03 BOOL  ; Spare
Last_Loaded_Recipe_Spare_Bits_WD4_bit4 D3024.04 BOOL  ; Spare
Last_Loaded_Recipe_Spare_Bits_WD4_bit5 D3024.05 BOOL  ; Spare
Last_Loaded_Recipe_Spare_Bits_WD4_bit6 D3024.06 BOOL  ; Spare
Last_Loaded_Recipe_Spare_Bits_WD4_bit7 D3024.07 BOOL  ; Spare
Last_Loaded_Recipe_Spare_Bits_WD4_bit8 D3024.08 BOOL  ; Spare
Last_Loaded_Recipe_Spare_Bits_WD4_bit9 D3024.09 BOOL  ; Spare
Last_Loaded_Recipe_Spare_Bits_WD5_bit0 D3025.00 BOOL  ; Spare
Last_Loaded_Recipe_Spare_Bits_WD5_bit1 D3025.01 BOOL  ; Spare
Last_Loaded_Recipe_Spare_Bits_WD5_bit10 D3025.10 BOOL  ; Spare
Last_Loaded_Recipe_Spare_Bits_WD5_bit11 D3025.11 BOOL  ; Spare
Last_Loaded_Recipe_Spare_Bits_WD5_bit12 D3025.12 BOOL  ; Spare
Last_Loaded_Recipe_Spare_Bits_WD5_bit13 D3025.13 BOOL  ; Spare
Last_Loaded_Recipe_Spare_Bits_WD5_bit14 D3025.14 BOOL  ; Spare
Last_Loaded_Recipe_Spare_Bits_WD5_bit15 D3025.15 BOOL  ; Spare
Last_Loaded_Recipe_Spare_Bits_WD5_bit2 D3025.02 BOOL  ; Spare
Last_Loaded_Recipe_Spare_Bits_WD5_bit3 D3025.03 BOOL  ; Spare
Last_Loaded_Recipe_Spare_Bits_WD5_bit4 D3025.04 BOOL  ; Spare
Last_Loaded_Recipe_Spare_Bits_WD5_bit5 D3025.05 BOOL  ; Spare
Last_Loaded_Recipe_Spare_Bits_WD5_bit6 D3025.06 BOOL  ; Spare
Last_Loaded_Recipe_Spare_Bits_WD5_bit7 D3025.07 BOOL  ; Spare
Last_Loaded_Recipe_Spare_Bits_WD5_bit8 D3025.08 BOOL  ; Spare
Last_Loaded_Recipe_Spare_Bits_WD5_bit9 D3025.09 BOOL  ; Spare
Last_Loaded_Recipe_Spare_Bits_WD6_bit0 D3026.00 BOOL  ; Spare
Last_Loaded_Recipe_Spare_Bits_WD6_bit1 D3026.01 BOOL  ; Spare
Last_Loaded_Recipe_Spare_Bits_WD6_bit10 D3026.10 BOOL  ; Spare
Last_Loaded_Recipe_Spare_Bits_WD6_bit11 D3026.11 BOOL  ; Spare
Last_Loaded_Recipe_Spare_Bits_WD6_bit12 D3026.12 BOOL  ; Spare
Last_Loaded_Recipe_Spare_Bits_WD6_bit13 D3026.13 BOOL  ; Spare
Last_Loaded_Recipe_Spare_Bits_WD6_bit14 D3026.14 BOOL  ; Spare
Last_Loaded_Recipe_Spare_Bits_WD6_bit15 D3026.15 BOOL  ; Spare
Last_Loaded_Recipe_Spare_Bits_WD6_bit2 D3026.02 BOOL  ; Spare
Last_Loaded_Recipe_Spare_Bits_WD6_bit3 D3026.03 BOOL  ; Spare
Last_Loaded_Recipe_Spare_Bits_WD6_bit4 D3026.04 BOOL  ; Spare
Last_Loaded_Recipe_Spare_Bits_WD6_bit5 D3026.05 BOOL  ; Spare
Last_Loaded_Recipe_Spare_Bits_WD6_bit6 D3026.06 BOOL  ; Spare
Last_Loaded_Recipe_Spare_Bits_WD6_bit7 D3026.07 BOOL  ; Spare
Last_Loaded_Recipe_Spare_Bits_WD6_bit8 D3026.08 BOOL  ; Spare
Last_Loaded_Recipe_Spare_Bits_WD6_bit9 D3026.09 BOOL  ; Spare
Last_Loaded_Recipe_Spare_Bits_WD7_bit0 D3027.00 BOOL  ; Spare
Last_Loaded_Recipe_Spare_Bits_WD7_bit1 D3027.01 BOOL  ; Spare
Last_Loaded_Recipe_Spare_Bits_WD7_bit10 D3027.10 BOOL  ; Spare
Last_Loaded_Recipe_Spare_Bits_WD7_bit11 D3027.11 BOOL  ; Spare
Last_Loaded_Recipe_Spare_Bits_WD7_bit12 D3027.12 BOOL  ; Spare
Last_Loaded_Recipe_Spare_Bits_WD7_bit13 D3027.13 BOOL  ; Spare
Last_Loaded_Recipe_Spare_Bits_WD7_bit14 D3027.14 BOOL  ; Spare
Last_Loaded_Recipe_Spare_Bits_WD7_bit15 D3027.15 BOOL  ; Spare
Last_Loaded_Recipe_Spare_Bits_WD7_bit2 D3027.02 BOOL  ; Spare
Last_Loaded_Recipe_Spare_Bits_WD7_bit3 D3027.03 BOOL  ; Spare
Last_Loaded_Recipe_Spare_Bits_WD7_bit4 D3027.04 BOOL  ; Spare
Last_Loaded_Recipe_Spare_Bits_WD7_bit5 D3027.05 BOOL  ; Spare
Last_Loaded_Recipe_Spare_Bits_WD7_bit6 D3027.06 BOOL  ; Spare
Last_Loaded_Recipe_Spare_Bits_WD7_bit7 D3027.07 BOOL  ; Spare
Last_Loaded_Recipe_Spare_Bits_WD7_bit8 D3027.08 BOOL  ; Spare
Last_Loaded_Recipe_Spare_Bits_WD7_bit9 D3027.09 BOOL  ; Spare
Last_Loaded_Recipe_Spare_Bits_WD8_bit0 D3028.00 BOOL  ; Spare
Last_Loaded_Recipe_Spare_Bits_WD8_bit1 D3028.01 BOOL  ; Spare
Last_Loaded_Recipe_Spare_Bits_WD8_bit10 D3028.10 BOOL  ; Spare
Last_Loaded_Recipe_Spare_Bits_WD8_bit11 D3028.11 BOOL  ; Spare
Last_Loaded_Recipe_Spare_Bits_WD8_bit12 D3028.12 BOOL  ; Spare
Last_Loaded_Recipe_Spare_Bits_WD8_bit13 D3028.13 BOOL  ; Spare
Last_Loaded_Recipe_Spare_Bits_WD8_bit14 D3028.14 BOOL  ; Spare
Last_Loaded_Recipe_Spare_Bits_WD8_bit15 D3028.15 BOOL  ; Spare
Last_Loaded_Recipe_Spare_Bits_WD8_bit2 D3028.02 BOOL  ; Spare
Last_Loaded_Recipe_Spare_Bits_WD8_bit3 D3028.03 BOOL  ; Spare
Last_Loaded_Recipe_Spare_Bits_WD8_bit4 D3028.04 BOOL  ; Spare
Last_Loaded_Recipe_Spare_Bits_WD8_bit5 D3028.05 BOOL  ; Spare
Last_Loaded_Recipe_Spare_Bits_WD8_bit6 D3028.06 BOOL  ; Spare
Last_Loaded_Recipe_Spare_Bits_WD8_bit7 D3028.07 BOOL  ; Spare
Last_Loaded_Recipe_Spare_Bits_WD8_bit8 D3028.08 BOOL  ; Spare
Last_Loaded_Recipe_Spare_Bits_WD8_bit9 D3028.09 BOOL  ; Spare
Last_Loaded_Recipe_Spare_UINT0 D3082 UINT
Last_Loaded_Recipe_Spare_UINT1 D3083 UINT
Last_Loaded_Recipe_Spare_UINT10 D3092 UINT
Last_Loaded_Recipe_Spare_UINT100 D3182 UINT
Last_Loaded_Recipe_Spare_UINT101 D3183 UINT
Last_Loaded_Recipe_Spare_UINT102 D3184 UINT
Last_Loaded_Recipe_Spare_UINT103 D3185 UINT
Last_Loaded_Recipe_Spare_UINT104 D3186 UINT
Last_Loaded_Recipe_Spare_UINT105 D3187 UINT
Last_Loaded_Recipe_Spare_UINT106 D3188 UINT
Last_Loaded_Recipe_Spare_UINT107 D3189 UINT
Last_Loaded_Recipe_Spare_UINT108 D3190 UINT
Last_Loaded_Recipe_Spare_UINT109 D3191 UINT
Last_Loaded_Recipe_Spare_UINT11 D3093 UINT
Last_Loaded_Recipe_Spare_UINT110 D3192 UINT
Last_Loaded_Recipe_Spare_UINT111 D3193 UINT
Last_Loaded_Recipe_Spare_UINT112 D3194 UINT
Last_Loaded_Recipe_Spare_UINT113 D3195 UINT
Last_Loaded_Recipe_Spare_UINT114 D3196 UINT
Last_Loaded_Recipe_Spare_UINT115 D3197 UINT
Last_Loaded_Recipe_Spare_UINT116 D3198 UINT
Last_Loaded_Recipe_Spare_UINT117 D3199 UINT
Last_Loaded_Recipe_Spare_UINT118 D3200 UINT
Last_Loaded_Recipe_Spare_UINT119 D3201 UINT
Last_Loaded_Recipe_Spare_UINT12 D3094 UINT
Last_Loaded_Recipe_Spare_UINT120 D3202 UINT
Last_Loaded_Recipe_Spare_UINT121 D3203 UINT
Last_Loaded_Recipe_Spare_UINT122 D3204 UINT
Last_Loaded_Recipe_Spare_UINT123 D3205 UINT
Last_Loaded_Recipe_Spare_UINT124 D3206 UINT
Last_Loaded_Recipe_Spare_UINT125 D3207 UINT
Last_Loaded_Recipe_Spare_UINT126 D3208 UINT
Last_Loaded_Recipe_Spare_UINT127 D3209 UINT
Last_Loaded_Recipe_Spare_UINT128 D3210 UINT
Last_Loaded_Recipe_Spare_UINT129 D3211 UINT
Last_Loaded_Recipe_Spare_UINT13 D3095 UINT
Last_Loaded_Recipe_Spare_UINT130 D3212 UINT
Last_Loaded_Recipe_Spare_UINT131 D3213 UINT
Last_Loaded_Recipe_Spare_UINT132 D3214 UINT
Last_Loaded_Recipe_Spare_UINT133 D3215 UINT
Last_Loaded_Recipe_Spare_UINT134 D3216 UINT
Last_Loaded_Recipe_Spare_UINT135 D3217 UINT
Last_Loaded_Recipe_Spare_UINT136 D3218 UINT
Last_Loaded_Recipe_Spare_UINT137 D3219 UINT
Last_Loaded_Recipe_Spare_UINT138 D3220 UINT
Last_Loaded_Recipe_Spare_UINT139 D3221 UINT
Last_Loaded_Recipe_Spare_UINT14 D3096 UINT
Last_Loaded_Recipe_Spare_UINT140 D3222 UINT
Last_Loaded_Recipe_Spare_UINT141 D3223 UINT
Last_Loaded_Recipe_Spare_UINT142 D3224 UINT
Last_Loaded_Recipe_Spare_UINT143 D3225 UINT
Last_Loaded_Recipe_Spare_UINT144 D3226 UINT
Last_Loaded_Recipe_Spare_UINT145 D3227 UINT
Last_Loaded_Recipe_Spare_UINT146 D3228 UINT
Last_Loaded_Recipe_Spare_UINT147 D3229 UINT
Last_Loaded_Recipe_Spare_UINT148 D3230 UINT
Last_Loaded_Recipe_Spare_UINT149 D3231 UINT
Last_Loaded_Recipe_Spare_UINT15 D3097 UINT
Last_Loaded_Recipe_Spare_UINT150 D3232 UINT
Last_Loaded_Recipe_Spare_UINT151 D3233 UINT
Last_Loaded_Recipe_Spare_UINT152 D3234 UINT
Last_Loaded_Recipe_Spare_UINT153 D3235 UINT
Last_Loaded_Recipe_Spare_UINT154 D3236 UINT
Last_Loaded_Recipe_Spare_UINT155 D3237 UINT
Last_Loaded_Recipe_Spare_UINT156 D3238 UINT
Last_Loaded_Recipe_Spare_UINT157 D3239 UINT
Last_Loaded_Recipe_Spare_UINT158 D3240 UINT
Last_Loaded_Recipe_Spare_UINT159 D3241 UINT
Last_Loaded_Recipe_Spare_UINT16 D3098 UINT
Last_Loaded_Recipe_Spare_UINT160 D3242 UINT
Last_Loaded_Recipe_Spare_UINT161 D3243 UINT
Last_Loaded_Recipe_Spare_UINT162 D3244 UINT
Last_Loaded_Recipe_Spare_UINT163 D3245 UINT
Last_Loaded_Recipe_Spare_UINT164 D3246 UINT
Last_Loaded_Recipe_Spare_UINT165 D3247 UINT
Last_Loaded_Recipe_Spare_UINT166 D3248 UINT
Last_Loaded_Recipe_Spare_UINT167 D3249 UINT
Last_Loaded_Recipe_Spare_UINT17 D3099 UINT
Last_Loaded_Recipe_Spare_UINT18 D3100 UINT
Last_Loaded_Recipe_Spare_UINT19 D3101 UINT
Last_Loaded_Recipe_Spare_UINT2 D3084 UINT
Last_Loaded_Recipe_Spare_UINT20 D3102 UINT
Last_Loaded_Recipe_Spare_UINT21 D3103 UINT
Last_Loaded_Recipe_Spare_UINT22 D3104 UINT
Last_Loaded_Recipe_Spare_UINT23 D3105 UINT
Last_Loaded_Recipe_Spare_UINT24 D3106 UINT
Last_Loaded_Recipe_Spare_UINT25 D3107 UINT
Last_Loaded_Recipe_Spare_UINT26 D3108 UINT
Last_Loaded_Recipe_Spare_UINT27 D3109 UINT
Last_Loaded_Recipe_Spare_UINT28 D3110 UINT
Last_Loaded_Recipe_Spare_UINT29 D3111 UINT
Last_Loaded_Recipe_Spare_UINT3 D3085 UINT
Last_Loaded_Recipe_Spare_UINT30 D3112 UINT
Last_Loaded_Recipe_Spare_UINT31 D3113 UINT
Last_Loaded_Recipe_Spare_UINT32 D3114 UINT
Last_Loaded_Recipe_Spare_UINT33 D3115 UINT
Last_Loaded_Recipe_Spare_UINT34 D3116 UINT
Last_Loaded_Recipe_Spare_UINT35 D3117 UINT
Last_Loaded_Recipe_Spare_UINT36 D3118 UINT
Last_Loaded_Recipe_Spare_UINT37 D3119 UINT
Last_Loaded_Recipe_Spare_UINT38 D3120 UINT
Last_Loaded_Recipe_Spare_UINT39 D3121 UINT
Last_Loaded_Recipe_Spare_UINT4 D3086 UINT
Last_Loaded_Recipe_Spare_UINT40 D3122 UINT
Last_Loaded_Recipe_Spare_UINT41 D3123 UINT
Last_Loaded_Recipe_Spare_UINT42 D3124 UINT
Last_Loaded_Recipe_Spare_UINT43 D3125 UINT
Last_Loaded_Recipe_Spare_UINT44 D3126 UINT
Last_Loaded_Recipe_Spare_UINT45 D3127 UINT
Last_Loaded_Recipe_Spare_UINT46 D3128 UINT
Last_Loaded_Recipe_Spare_UINT47 D3129 UINT
Last_Loaded_Recipe_Spare_UINT48 D3130 UINT
Last_Loaded_Recipe_Spare_UINT49 D3131 UINT
Last_Loaded_Recipe_Spare_UINT5 D3087 UINT
Last_Loaded_Recipe_Spare_UINT50 D3132 UINT
Last_Loaded_Recipe_Spare_UINT51 D3133 UINT
Last_Loaded_Recipe_Spare_UINT52 D3134 UINT
Last_Loaded_Recipe_Spare_UINT53 D3135 UINT
Last_Loaded_Recipe_Spare_UINT54 D3136 UINT
Last_Loaded_Recipe_Spare_UINT55 D3137 UINT
Last_Loaded_Recipe_Spare_UINT56 D3138 UINT
Last_Loaded_Recipe_Spare_UINT57 D3139 UINT
Last_Loaded_Recipe_Spare_UINT58 D3140 UINT
Last_Loaded_Recipe_Spare_UINT59 D3141 UINT
Last_Loaded_Recipe_Spare_UINT6 D3088 UINT
Last_Loaded_Recipe_Spare_UINT60 D3142 UINT
Last_Loaded_Recipe_Spare_UINT61 D3143 UINT
Last_Loaded_Recipe_Spare_UINT62 D3144 UINT
Last_Loaded_Recipe_Spare_UINT63 D3145 UINT
Last_Loaded_Recipe_Spare_UINT64 D3146 UINT
Last_Loaded_Recipe_Spare_UINT65 D3147 UINT
Last_Loaded_Recipe_Spare_UINT66 D3148 UINT
Last_Loaded_Recipe_Spare_UINT67 D3149 UINT
Last_Loaded_Recipe_Spare_UINT68 D3150 UINT
Last_Loaded_Recipe_Spare_UINT69 D3151 UINT
Last_Loaded_Recipe_Spare_UINT7 D3089 UINT
Last_Loaded_Recipe_Spare_UINT70 D3152 UINT
Last_Loaded_Recipe_Spare_UINT71 D3153 UINT
Last_Loaded_Recipe_Spare_UINT72 D3154 UINT
Last_Loaded_Recipe_Spare_UINT73 D3155 UINT
Last_Loaded_Recipe_Spare_UINT74 D3156 UINT
Last_Loaded_Recipe_Spare_UINT75 D3157 UINT
Last_Loaded_Recipe_Spare_UINT76 D3158 UINT
Last_Loaded_Recipe_Spare_UINT77 D3159 UINT
Last_Loaded_Recipe_Spare_UINT78 D3160 UINT
Last_Loaded_Recipe_Spare_UINT79 D3161 UINT
Last_Loaded_Recipe_Spare_UINT8 D3090 UINT
Last_Loaded_Recipe_Spare_UINT80 D3162 UINT
Last_Loaded_Recipe_Spare_UINT81 D3163 UINT
Last_Loaded_Recipe_Spare_UINT82 D3164 UINT
Last_Loaded_Recipe_Spare_UINT83 D3165 UINT
Last_Loaded_Recipe_Spare_UINT84 D3166 UINT
Last_Loaded_Recipe_Spare_UINT85 D3167 UINT
Last_Loaded_Recipe_Spare_UINT86 D3168 UINT
Last_Loaded_Recipe_Spare_UINT87 D3169 UINT
Last_Loaded_Recipe_Spare_UINT88 D3170 UINT
Last_Loaded_Recipe_Spare_UINT89 D3171 UINT
Last_Loaded_Recipe_Spare_UINT9 D3091 UINT
Last_Loaded_Recipe_Spare_UINT90 D3172 UINT
Last_Loaded_Recipe_Spare_UINT91 D3173 UINT
Last_Loaded_Recipe_Spare_UINT92 D3174 UINT
Last_Loaded_Recipe_Spare_UINT93 D3175 UINT
Last_Loaded_Recipe_Spare_UINT94 D3176 UINT
Last_Loaded_Recipe_Spare_UINT95 D3177 UINT
Last_Loaded_Recipe_Spare_UINT96 D3178 UINT
Last_Loaded_Recipe_Spare_UINT97 D3179 UINT
Last_Loaded_Recipe_Spare_UINT98 D3180 UINT
Last_Loaded_Recipe_Spare_UINT99 D3181 UINT
Last_Loaded_Recipe_Stale_Film_Time D3078 UINT
Last_Loaded_Recipe_Temp_Setpoint D3030 UINT  ; Tool temperature setpoint
Last_Loaded_Recipe_Tool_Position D3068 UINT
Last_Loaded_Recipe_Top_Vacuum_Delay D3035 UINT
Last_Loaded_Recipe_Tray_Position D3062 UINT
Last_Loaded_Recipe_Tray_Settle_Time D3056 UINT
Last_Loaded_Recipe_Tray_Stop_Delay D3053 UINT
Last_Loaded_Recipe_Upstream_Off_Delay D3061 UINT
Last_Loaded_Recipe_Upstream_On_Delay D3060 UINT
Last_Loaded_Recipe_VAC_Type D3020.00 BOOL  ; Vac type - ON = Pressure, OFF = Time
Last_Loaded_Recipe_Vacuum_Duration D3037 UINT
Last_Loaded_Recipe_Vacuum_Extra_Time D3039 UINT
Last_Loaded_Recipe_Vacuum_Pressure_SP D3038 UINT
Last_Loaded_Recipe_Vent_Bottom_Delay D3044 UINT
Last_Loaded_Recipe_Vent_Duration D3045 UINT
Last_Loaded_Recipe_Vent_Pressure_SP D3046 UINT
Last_Loaded_Recipe_Vent_Top_Delay D3043 UINT
Last_Loaded_Recipe_Vent_Type D3020.02 BOOL  ; Vent type - ON = Pressure, OFF = Time
Last_Low_Tolerance D932 UINT
Last_Max_SP D928 UINT
Last_Number_of_Trays D516 UINT  ; Contains the last number of trays
Last_Overtemp_SP D930 UINT
Last_Setpoint D926 UINT
Last_Sleep_Mode_Temp D936 UINT
Lifetime_Cycles D804 DINT  ; Lifetime Cycle count
Lift_Down_Decel_Off_Delay T0214 TIMER  ; Off delay for lift down decel
Lift_Down_Delay T0226 TIMER  ; Delay Lwr Tool Down for lowering
Lift_Down_Off_Delay T0212 TIMER  ; Off delay for lift down
Lift_Down_WD_Fault W150.09 BOOL  ; Watchdog Timer Fault
Lift_Down_WD_Timer T0138 TIMER  ; Watchdog Timer
Lift_Up_Decel_Off_Delay T0213 TIMER  ; Off delay for lift up decel
Lift_Up_Off_Delay T0211 TIMER  ; Off delay for lift up
Lift_Up_Refresh T0225 TIMER  ; Energize Lwr Tool Up before lowering
Lift_Up_WD_Fault W150.08 BOOL  ; Watchdog Timer Fault
Lift_Up_WD_Timer T0137 TIMER  ; Watchdog Timer
Loaded_Recipe_Advance_Accel_Percent D71 UINT
Loaded_Recipe_Advance_Decel_Percent D72 UINT
Loaded_Recipe_Advance_Time D69 UINT
Loaded_Recipe_Advance_Velocity_Percent D70 UINT
Loaded_Recipe_Auto_gas_offset D110 UINT  ; Offset Scaled Gas result
Loaded_Recipe_Bottom_Vacuum_Delay D36 UINT
Loaded_Recipe_Conveyor_gate_time D113 UINT  ; Time to see tray before stopping upstream
Loaded_Recipe_Cycle_Type D29 UINT  ; Cycle type selection (Flat, Map, Simultaneous, VSP)
Loaded_Recipe_Dancing_Stop D58 UINT
Loaded_Recipe_Default_Gas_setting D114 UINT  ; Default gas time for autogassing
Loaded_Recipe_Delay_tray_measurement D111 UINT  ; Delay tray measurement time
Loaded_Recipe_Feed_Delay_After_Adv D52 UINT
Loaded_Recipe_Film_Feed_Accel D76 UINT
Loaded_Recipe_Film_Feed_Accel_clear D76 UINT
Loaded_Recipe_Film_Feed_Accel_reg D248 UINT
Loaded_Recipe_Film_Feed_Decel D77 UINT
Loaded_Recipe_Film_Feed_Decel_clear D77 UINT
Loaded_Recipe_Film_Feed_Decel_reg D249 UINT
Loaded_Recipe_Film_Feed_Velocity D75 UINT
Loaded_Recipe_Film_Feed_Velocity_Reg D247 UINT
Loaded_Recipe_Film_Feed_Velocity_clear D75 UINT
Loaded_Recipe_Film_Jog_Accel D80 UINT
Loaded_Recipe_Film_Jog_Decel D81 UINT
Loaded_Recipe_Film_Jog_Velocity D79 UINT
Loaded_Recipe_Film_Length D31 UINT  ; Film length to feed
Loaded_Recipe_Gas_Delay D40 UINT
Loaded_Recipe_Gas_Duration D41 UINT
Loaded_Recipe_Gas_Pressure_SP D42 UINT
Loaded_Recipe_Gas_Type D20.01 BOOL  ; Gas type - ON = Pressure, OFF = Time
Loaded_Recipe_Grip_Open_Delay D67 UINT
Loaded_Recipe_Gripper_ADV_Delay D57 UINT
Loaded_Recipe_Gripper_Close_Delay D50 UINT
Loaded_Recipe_Infeed_Gate_Eye_Debounce D55 UINT
Loaded_Recipe_Infeed_speed D34 UINT  ; Infeed speed setting
Loaded_Recipe_LP1_CP D85 UINT  ; LP1 CP
Loaded_Recipe_LP1_D D84 UINT
Loaded_Recipe_LP1_I D83 UINT
Loaded_Recipe_LP1_P D82 UINT
Loaded_Recipe_LP2_CP D89 UINT
Loaded_Recipe_LP2_D D88 UINT
Loaded_Recipe_LP2_I D87 UINT
Loaded_Recipe_LP2_P D86 UINT
Loaded_Recipe_LP3_CP D93 UINT
Loaded_Recipe_LP3_D D92 UINT
Loaded_Recipe_LP3_I D91 UINT
Loaded_Recipe_LP3_P D90 UINT
Loaded_Recipe_LP4_CP D97 UINT  ; LP4CP
Loaded_Recipe_LP4_D D96 UINT
Loaded_Recipe_LP4_I D95 UINT
Loaded_Recipe_LP4_P D94 UINT
Loaded_Recipe_LP5_CP D101 UINT
Loaded_Recipe_LP5_D D100 UINT
Loaded_Recipe_LP5_I D99 UINT
Loaded_Recipe_LP5_P D98 UINT
Loaded_Recipe_LP6_CP D105 UINT
Loaded_Recipe_LP6_D D104 UINT
Loaded_Recipe_LP6_I D103 UINT
Loaded_Recipe_LP6_P D102 UINT
Loaded_Recipe_Lift_Decel D73 UINT
Loaded_Recipe_Lost_Tray_Reset_Delay D54 UINT
Loaded_Recipe_Lower_Decel D74 UINT
Loaded_Recipe_Maximum_auto_gas D109 UINT  ; Maximum setpoint for scaling
Loaded_Recipe_Measurement_Infeed D106 UINT  ; Time for tray measurement at Infeed Gate
Loaded_Recipe_Measurement_Stop_2 D107 UINT  ; Time for tray measurement at Stop 2
Loaded_Recipe_Min_tray_size D115 UINT  ; minimum height of tray
Loaded_Recipe_Minimum_auto_gas D108 UINT  ; Minimum setpoint for scaling
Loaded_Recipe_Motion_Setting_from_Time D20.05 BOOL  ; Chooses time setting or vel, accel and decel settings
Loaded_Recipe_Name D0 STRING[38]  ; Job name for Recipe 0
Loaded_Recipe_Number D19 CHANNEL  ; Recipe Number (0 - 99)
Loaded_Recipe_Number_of_Trays D59 UINT  ; # of trays in tool
Loaded_Recipe_REV_Yank D20.03 BOOL  ; On if reverse yank enabled for film
Loaded_Recipe_Reg_Offset D33 UINT  ; Registration Offset
Loaded_Recipe_Reg_enable D20.04 BOOL  ; On if registration enabled for film
Loaded_Recipe_Return_Accel_Percent D65 UINT
Loaded_Recipe_Return_Decel_Percent D66 UINT
Loaded_Recipe_Return_Time D63 UINT
Loaded_Recipe_Return_Velocity_Percent D64 UINT
Loaded_Recipe_Rev_Yank_Dist D32 UINT  ; Reverse Yank Distance
Loaded_Recipe_Rewind_On_Delay D51 UINT
Loaded_Recipe_Seal_Cool D49 UINT
Loaded_Recipe_Seal_Delay D47 UINT
Loaded_Recipe_Seal_Duration D48 UINT
Loaded_Recipe_Slow_Down_Length D244 UINT
Loaded_Recipe_Spare_Bits_WD0_bit10 D20.10 BOOL  ; Spare
Loaded_Recipe_Spare_Bits_WD0_bit11 D20.11 BOOL  ; Spare
Loaded_Recipe_Spare_Bits_WD0_bit12 D20.12 BOOL  ; Spare
Loaded_Recipe_Spare_Bits_WD0_bit13 D20.13 BOOL  ; Spare
Loaded_Recipe_Spare_Bits_WD0_bit14 D20.14 BOOL  ; Spare
Loaded_Recipe_Spare_Bits_WD0_bit15 D20.15 BOOL  ; Spare
Loaded_Recipe_Spare_Bits_WD0_bit8 D20.08 BOOL  ; Spare
Loaded_Recipe_Spare_Bits_WD0_bit9 D20.09 BOOL  ; Spare
Loaded_Recipe_Spare_Bits_WD1_bit0 D21.00 BOOL  ; Spare
Loaded_Recipe_Spare_Bits_WD1_bit1 D21.01 BOOL  ; Spare
Loaded_Recipe_Spare_Bits_WD1_bit10 D21.10 BOOL  ; Spare
Loaded_Recipe_Spare_Bits_WD1_bit11 D21.11 BOOL  ; Spare
Loaded_Recipe_Spare_Bits_WD1_bit12 D21.12 BOOL  ; Spare
Loaded_Recipe_Spare_Bits_WD1_bit13 D21.13 BOOL  ; Spare
Loaded_Recipe_Spare_Bits_WD1_bit14 D21.14 BOOL  ; Spare
Loaded_Recipe_Spare_Bits_WD1_bit15 D21.15 BOOL  ; Spare
Loaded_Recipe_Spare_Bits_WD1_bit2 D21.02 BOOL  ; Spare
Loaded_Recipe_Spare_Bits_WD1_bit3 D21.03 BOOL  ; Spare
Loaded_Recipe_Spare_Bits_WD1_bit4 D21.04 BOOL  ; Spare
Loaded_Recipe_Spare_Bits_WD1_bit5 D21.05 BOOL  ; Spare
Loaded_Recipe_Spare_Bits_WD1_bit6 D21.06 BOOL  ; Spare
Loaded_Recipe_Spare_Bits_WD1_bit7 D21.07 BOOL  ; Spare
Loaded_Recipe_Spare_Bits_WD1_bit8 D21.08 BOOL  ; Spare
Loaded_Recipe_Spare_Bits_WD1_bit9 D21.09 BOOL  ; Spare
Loaded_Recipe_Spare_Bits_WD2_bit0 D22.00 BOOL  ; Spare
Loaded_Recipe_Spare_Bits_WD2_bit1 D22.01 BOOL  ; Spare
Loaded_Recipe_Spare_Bits_WD2_bit10 D22.10 BOOL  ; Spare
Loaded_Recipe_Spare_Bits_WD2_bit11 D22.11 BOOL  ; Spare
Loaded_Recipe_Spare_Bits_WD2_bit12 D22.12 BOOL  ; Spare
Loaded_Recipe_Spare_Bits_WD2_bit13 D22.13 BOOL  ; Spare
Loaded_Recipe_Spare_Bits_WD2_bit14 D22.14 BOOL  ; Spare
Loaded_Recipe_Spare_Bits_WD2_bit15 D22.15 BOOL  ; Spare
Loaded_Recipe_Spare_Bits_WD2_bit2 D22.02 BOOL  ; Spare
Loaded_Recipe_Spare_Bits_WD2_bit3 D22.03 BOOL  ; Spare
Loaded_Recipe_Spare_Bits_WD2_bit4 D22.04 BOOL  ; Spare
Loaded_Recipe_Spare_Bits_WD2_bit5 D22.05 BOOL  ; Spare
Loaded_Recipe_Spare_Bits_WD2_bit6 D22.06 BOOL  ; Spare
Loaded_Recipe_Spare_Bits_WD2_bit7 D22.07 BOOL  ; Spare
Loaded_Recipe_Spare_Bits_WD2_bit8 D22.08 BOOL  ; Spare
Loaded_Recipe_Spare_Bits_WD2_bit9 D22.09 BOOL  ; Spare
Loaded_Recipe_Spare_Bits_WD3_bit0 D23.00 BOOL  ; Spare
Loaded_Recipe_Spare_Bits_WD3_bit1 D23.01 BOOL  ; Spare
Loaded_Recipe_Spare_Bits_WD3_bit10 D23.10 BOOL  ; Spare
Loaded_Recipe_Spare_Bits_WD3_bit11 D23.11 BOOL  ; Spare
Loaded_Recipe_Spare_Bits_WD3_bit12 D23.12 BOOL  ; Spare
Loaded_Recipe_Spare_Bits_WD3_bit13 D23.13 BOOL  ; Spare
Loaded_Recipe_Spare_Bits_WD3_bit14 D23.14 BOOL  ; Spare
Loaded_Recipe_Spare_Bits_WD3_bit15 D23.15 BOOL  ; Spare
Loaded_Recipe_Spare_Bits_WD3_bit2 D23.02 BOOL  ; Spare
Loaded_Recipe_Spare_Bits_WD3_bit3 D23.03 BOOL  ; Spare
Loaded_Recipe_Spare_Bits_WD3_bit4 D23.04 BOOL  ; Spare
Loaded_Recipe_Spare_Bits_WD3_bit5 D23.05 BOOL  ; Spare
Loaded_Recipe_Spare_Bits_WD3_bit6 D23.06 BOOL  ; Spare
Loaded_Recipe_Spare_Bits_WD3_bit7 D23.07 BOOL  ; Spare
Loaded_Recipe_Spare_Bits_WD3_bit8 D23.08 BOOL  ; Spare
Loaded_Recipe_Spare_Bits_WD3_bit9 D23.09 BOOL  ; Spare
Loaded_Recipe_Spare_Bits_WD4_bit0 D24.00 BOOL  ; Spare
Loaded_Recipe_Spare_Bits_WD4_bit1 D24.01 BOOL  ; Spare
Loaded_Recipe_Spare_Bits_WD4_bit10 D24.10 BOOL  ; Spare
Loaded_Recipe_Spare_Bits_WD4_bit11 D24.11 BOOL  ; Spare
Loaded_Recipe_Spare_Bits_WD4_bit12 D24.12 BOOL  ; Spare
Loaded_Recipe_Spare_Bits_WD4_bit13 D24.13 BOOL  ; Spare
Loaded_Recipe_Spare_Bits_WD4_bit14 D24.14 BOOL  ; Spare
Loaded_Recipe_Spare_Bits_WD4_bit15 D24.15 BOOL  ; Spare
Loaded_Recipe_Spare_Bits_WD4_bit2 D24.02 BOOL  ; Spare
Loaded_Recipe_Spare_Bits_WD4_bit3 D24.03 BOOL  ; Spare
Loaded_Recipe_Spare_Bits_WD4_bit4 D24.04 BOOL  ; Spare
Loaded_Recipe_Spare_Bits_WD4_bit5 D24.05 BOOL  ; Spare
Loaded_Recipe_Spare_Bits_WD4_bit6 D24.06 BOOL  ; Spare
Loaded_Recipe_Spare_Bits_WD4_bit7 D24.07 BOOL  ; Spare
Loaded_Recipe_Spare_Bits_WD4_bit8 D24.08 BOOL  ; Spare
Loaded_Recipe_Spare_Bits_WD4_bit9 D24.09 BOOL  ; Spare
Loaded_Recipe_Spare_Bits_WD5_bit0 D25.00 BOOL  ; Spare
Loaded_Recipe_Spare_Bits_WD5_bit1 D25.01 BOOL  ; Spare
Loaded_Recipe_Spare_Bits_WD5_bit10 D25.10 BOOL  ; Spare
Loaded_Recipe_Spare_Bits_WD5_bit11 D25.11 BOOL  ; Spare
Loaded_Recipe_Spare_Bits_WD5_bit12 D25.12 BOOL  ; Spare
Loaded_Recipe_Spare_Bits_WD5_bit13 D25.13 BOOL  ; Spare
Loaded_Recipe_Spare_Bits_WD5_bit14 D25.14 BOOL  ; Spare
Loaded_Recipe_Spare_Bits_WD5_bit15 D25.15 BOOL  ; Spare
Loaded_Recipe_Spare_Bits_WD5_bit2 D25.02 BOOL  ; Spare
Loaded_Recipe_Spare_Bits_WD5_bit3 D25.03 BOOL  ; Spare
Loaded_Recipe_Spare_Bits_WD5_bit4 D25.04 BOOL  ; Spare
Loaded_Recipe_Spare_Bits_WD5_bit5 D25.05 BOOL  ; Spare
Loaded_Recipe_Spare_Bits_WD5_bit6 D25.06 BOOL  ; Spare
Loaded_Recipe_Spare_Bits_WD5_bit7 D25.07 BOOL  ; Spare
Loaded_Recipe_Spare_Bits_WD5_bit8 D25.08 BOOL  ; Spare
Loaded_Recipe_Spare_Bits_WD5_bit9 D25.09 BOOL  ; Spare
Loaded_Recipe_Spare_Bits_WD6_bit0 D26.00 BOOL  ; Spare
Loaded_Recipe_Spare_Bits_WD6_bit1 D26.01 BOOL  ; Spare
Loaded_Recipe_Spare_Bits_WD6_bit10 D26.10 BOOL  ; Spare
Loaded_Recipe_Spare_Bits_WD6_bit11 D26.11 BOOL  ; Spare
Loaded_Recipe_Spare_Bits_WD6_bit12 D26.12 BOOL  ; Spare
Loaded_Recipe_Spare_Bits_WD6_bit13 D26.13 BOOL  ; Spare
Loaded_Recipe_Spare_Bits_WD6_bit14 D26.14 BOOL  ; Spare
Loaded_Recipe_Spare_Bits_WD6_bit15 D26.15 BOOL  ; Spare
Loaded_Recipe_Spare_Bits_WD6_bit2 D26.02 BOOL  ; Spare
Loaded_Recipe_Spare_Bits_WD6_bit3 D26.03 BOOL  ; Spare
Loaded_Recipe_Spare_Bits_WD6_bit4 D26.04 BOOL  ; Spare
Loaded_Recipe_Spare_Bits_WD6_bit5 D26.05 BOOL  ; Spare
Loaded_Recipe_Spare_Bits_WD6_bit6 D26.06 BOOL  ; Spare
Loaded_Recipe_Spare_Bits_WD6_bit7 D26.07 BOOL  ; Spare
Loaded_Recipe_Spare_Bits_WD6_bit8 D26.08 BOOL  ; Spare
Loaded_Recipe_Spare_Bits_WD6_bit9 D26.09 BOOL  ; Spare
Loaded_Recipe_Spare_Bits_WD7_bit0 D27.00 BOOL  ; Spare
Loaded_Recipe_Spare_Bits_WD7_bit1 D27.01 BOOL  ; Spare
Loaded_Recipe_Spare_Bits_WD7_bit10 D27.10 BOOL  ; Spare
Loaded_Recipe_Spare_Bits_WD7_bit11 D27.11 BOOL  ; Spare
Loaded_Recipe_Spare_Bits_WD7_bit12 D27.12 BOOL  ; Spare
Loaded_Recipe_Spare_Bits_WD7_bit13 D27.13 BOOL  ; Spare
Loaded_Recipe_Spare_Bits_WD7_bit14 D27.14 BOOL  ; Spare
Loaded_Recipe_Spare_Bits_WD7_bit15 D27.15 BOOL  ; Spare
Loaded_Recipe_Spare_Bits_WD7_bit2 D27.02 BOOL  ; Spare
Loaded_Recipe_Spare_Bits_WD7_bit3 D27.03 BOOL  ; Spare
Loaded_Recipe_Spare_Bits_WD7_bit4 D27.04 BOOL  ; Spare
Loaded_Recipe_Spare_Bits_WD7_bit5 D27.05 BOOL  ; Spare
Loaded_Recipe_Spare_Bits_WD7_bit6 D27.06 BOOL  ; Spare
Loaded_Recipe_Spare_Bits_WD7_bit7 D27.07 BOOL  ; Spare
Loaded_Recipe_Spare_Bits_WD7_bit8 D27.08 BOOL  ; Spare
Loaded_Recipe_Spare_Bits_WD7_bit9 D27.09 BOOL  ; Spare
Loaded_Recipe_Spare_Bits_WD8_bit0 D28.00 BOOL  ; Spare
Loaded_Recipe_Spare_Bits_WD8_bit1 D28.01 BOOL  ; Spare
Loaded_Recipe_Spare_Bits_WD8_bit10 D28.10 BOOL  ; Spare
Loaded_Recipe_Spare_Bits_WD8_bit11 D28.11 BOOL  ; Spare
Loaded_Recipe_Spare_Bits_WD8_bit12 D28.12 BOOL  ; Spare
Loaded_Recipe_Spare_Bits_WD8_bit13 D28.13 BOOL  ; Spare
Loaded_Recipe_Spare_Bits_WD8_bit14 D28.14 BOOL  ; Spare
Loaded_Recipe_Spare_Bits_WD8_bit2 D28.02 BOOL  ; Spare
Loaded_Recipe_Spare_Bits_WD8_bit3 D28.03 BOOL  ; Spare
Loaded_Recipe_Spare_Bits_WD8_bit4 D28.04 BOOL  ; Spare
Loaded_Recipe_Spare_Bits_WD8_bit5 D28.05 BOOL  ; Spare
Loaded_Recipe_Spare_Bits_WD8_bit6 D28.06 BOOL  ; Spare
Loaded_Recipe_Spare_Bits_WD8_bit7 D28.07 BOOL  ; Spare
Loaded_Recipe_Spare_Bits_WD8_bit8 D28.08 BOOL  ; Spare
Loaded_Recipe_Spare_Bits_WD8_bit9 D28.09 BOOL  ; Spare
Loaded_Recipe_Spare_UINT100 D182 UINT
Loaded_Recipe_Spare_UINT101 D183 UINT
Loaded_Recipe_Spare_UINT102 D184 UINT
Loaded_Recipe_Spare_UINT103 D185 UINT
Loaded_Recipe_Spare_UINT104 D186 UINT
Loaded_Recipe_Spare_UINT105 D187 UINT
Loaded_Recipe_Spare_UINT106 D188 UINT
Loaded_Recipe_Spare_UINT107 D189 UINT
Loaded_Recipe_Spare_UINT108 D190 UINT
Loaded_Recipe_Spare_UINT109 D191 UINT
Loaded_Recipe_Spare_UINT110 D192 UINT
Loaded_Recipe_Spare_UINT111 D193 UINT
Loaded_Recipe_Spare_UINT112 D194 UINT
Loaded_Recipe_Spare_UINT113 D195 UINT
Loaded_Recipe_Spare_UINT114 D196 UINT
Loaded_Recipe_Spare_UINT115 D197 UINT
Loaded_Recipe_Spare_UINT116 D198 UINT
Loaded_Recipe_Spare_UINT117 D199 UINT
Loaded_Recipe_Spare_UINT118 D200 UINT
Loaded_Recipe_Spare_UINT119 D201 UINT
Loaded_Recipe_Spare_UINT120 D202 UINT
Loaded_Recipe_Spare_UINT121 D203 UINT
Loaded_Recipe_Spare_UINT122 D204 UINT
Loaded_Recipe_Spare_UINT123 D205 UINT
Loaded_Recipe_Spare_UINT124 D206 UINT
Loaded_Recipe_Spare_UINT125 D207 UINT
Loaded_Recipe_Spare_UINT126 D208 UINT
Loaded_Recipe_Spare_UINT127 D209 UINT
Loaded_Recipe_Spare_UINT128 D210 UINT
Loaded_Recipe_Spare_UINT129 D211 UINT
Loaded_Recipe_Spare_UINT130 D212 UINT
Loaded_Recipe_Spare_UINT131 D213 UINT
Loaded_Recipe_Spare_UINT132 D214 UINT
Loaded_Recipe_Spare_UINT133 D215 UINT
Loaded_Recipe_Spare_UINT134 D216 UINT
Loaded_Recipe_Spare_UINT135 D217 UINT
Loaded_Recipe_Spare_UINT136 D218 UINT
Loaded_Recipe_Spare_UINT137 D219 UINT
Loaded_Recipe_Spare_UINT138 D220 UINT
Loaded_Recipe_Spare_UINT139 D221 UINT
Loaded_Recipe_Spare_UINT140 D222 UINT
Loaded_Recipe_Spare_UINT141 D223 UINT
Loaded_Recipe_Spare_UINT142 D224 UINT
Loaded_Recipe_Spare_UINT143 D225 UINT
Loaded_Recipe_Spare_UINT144 D226 UINT
Loaded_Recipe_Spare_UINT145 D227 UINT
Loaded_Recipe_Spare_UINT146 D228 UINT
Loaded_Recipe_Spare_UINT147 D229 UINT
Loaded_Recipe_Spare_UINT148 D230 UINT
Loaded_Recipe_Spare_UINT149 D231 UINT
Loaded_Recipe_Spare_UINT150 D232 UINT
Loaded_Recipe_Spare_UINT151 D233 UINT
Loaded_Recipe_Spare_UINT152 D234 UINT
Loaded_Recipe_Spare_UINT153 D235 UINT
Loaded_Recipe_Spare_UINT154 D236 UINT
Loaded_Recipe_Spare_UINT155 D237 UINT
Loaded_Recipe_Spare_UINT156 D238 UINT
Loaded_Recipe_Spare_UINT157 D239 UINT
Loaded_Recipe_Spare_UINT158 D240 UINT
Loaded_Recipe_Spare_UINT159 D241 UINT
Loaded_Recipe_Spare_UINT160 D242 UINT
Loaded_Recipe_Spare_UINT161 D243 UINT
Loaded_Recipe_Spare_UINT162 D244 UINT
Loaded_Recipe_Spare_UINT163 D245 UINT
Loaded_Recipe_Spare_UINT164 D246 UINT
Loaded_Recipe_Spare_UINT165 D247 UINT
Loaded_Recipe_Spare_UINT166 D248 UINT
Loaded_Recipe_Spare_UINT167 D249 UINT
Loaded_Recipe_Spare_UINT27 D109 UINT
Loaded_Recipe_Spare_UINT28 D110 UINT
Loaded_Recipe_Spare_UINT29 D111 UINT
Loaded_Recipe_Spare_UINT30 D112 UINT
Loaded_Recipe_Spare_UINT31 D113 UINT
Loaded_Recipe_Spare_UINT32 D114 UINT
Loaded_Recipe_Spare_UINT33 D115 UINT
Loaded_Recipe_Spare_UINT34 D116 UINT
Loaded_Recipe_Spare_UINT35 D117 UINT
Loaded_Recipe_Spare_UINT36 D118 UINT
Loaded_Recipe_Spare_UINT37 D119 UINT
Loaded_Recipe_Spare_UINT38 D120 UINT
Loaded_Recipe_Spare_UINT39 D121 UINT
Loaded_Recipe_Spare_UINT40 D122 UINT
Loaded_Recipe_Spare_UINT41 D123 UINT
Loaded_Recipe_Spare_UINT42 D124 UINT
Loaded_Recipe_Spare_UINT43 D125 UINT
Loaded_Recipe_Spare_UINT44 D126 UINT
Loaded_Recipe_Spare_UINT45 D127 UINT
Loaded_Recipe_Spare_UINT46 D128 UINT
Loaded_Recipe_Spare_UINT47 D129 UINT
Loaded_Recipe_Spare_UINT48 D130 UINT
Loaded_Recipe_Spare_UINT49 D131 UINT
Loaded_Recipe_Spare_UINT50 D132 UINT
Loaded_Recipe_Spare_UINT51 D133 UINT
Loaded_Recipe_Spare_UINT52 D134 UINT
Loaded_Recipe_Spare_UINT53 D135 UINT
Loaded_Recipe_Spare_UINT54 D136 UINT
Loaded_Recipe_Spare_UINT55 D137 UINT
Loaded_Recipe_Spare_UINT56 D138 UINT
Loaded_Recipe_Spare_UINT57 D139 UINT
Loaded_Recipe_Spare_UINT58 D140 UINT
Loaded_Recipe_Spare_UINT59 D141 UINT
Loaded_Recipe_Spare_UINT60 D142 UINT
Loaded_Recipe_Spare_UINT61 D143 UINT
Loaded_Recipe_Spare_UINT62 D144 UINT
Loaded_Recipe_Spare_UINT63 D145 UINT
Loaded_Recipe_Spare_UINT64 D146 UINT
Loaded_Recipe_Spare_UINT65 D147 UINT
Loaded_Recipe_Spare_UINT66 D148 UINT
Loaded_Recipe_Spare_UINT67 D149 UINT
Loaded_Recipe_Spare_UINT68 D150 UINT
Loaded_Recipe_Spare_UINT69 D151 UINT
Loaded_Recipe_Spare_UINT70 D152 UINT
Loaded_Recipe_Spare_UINT71 D153 UINT
Loaded_Recipe_Spare_UINT72 D154 UINT
Loaded_Recipe_Spare_UINT73 D155 UINT
Loaded_Recipe_Spare_UINT74 D156 UINT
Loaded_Recipe_Spare_UINT75 D157 UINT
Loaded_Recipe_Spare_UINT76 D158 UINT
Loaded_Recipe_Spare_UINT77 D159 UINT
Loaded_Recipe_Spare_UINT78 D160 UINT
Loaded_Recipe_Spare_UINT79 D161 UINT
Loaded_Recipe_Spare_UINT80 D162 UINT
Loaded_Recipe_Spare_UINT81 D163 UINT
Loaded_Recipe_Spare_UINT82 D164 UINT
Loaded_Recipe_Spare_UINT83 D165 UINT
Loaded_Recipe_Spare_UINT84 D166 UINT
Loaded_Recipe_Spare_UINT85 D167 UINT
Loaded_Recipe_Spare_UINT86 D168 UINT
Loaded_Recipe_Spare_UINT87 D169 UINT
Loaded_Recipe_Spare_UINT88 D170 UINT
Loaded_Recipe_Spare_UINT89 D171 UINT
Loaded_Recipe_Spare_UINT90 D172 UINT
Loaded_Recipe_Spare_UINT91 D173 UINT
Loaded_Recipe_Spare_UINT92 D174 UINT
Loaded_Recipe_Spare_UINT93 D175 UINT
Loaded_Recipe_Spare_UINT94 D176 UINT
Loaded_Recipe_Spare_UINT95 D177 UINT
Loaded_Recipe_Spare_UINT96 D178 UINT
Loaded_Recipe_Spare_UINT97 D179 UINT
Loaded_Recipe_Spare_UINT98 D180 UINT
Loaded_Recipe_Spare_UINT99 D181 UINT
Loaded_Recipe_Stale_Film_Time D78 UINT
Loaded_Recipe_Temp_Setpoint D30 UINT  ; Tool temperature setpoint
Loaded_Recipe_Tool_Position D68 UINT
Loaded_Recipe_Top_Vacuum_Delay D35 UINT
Loaded_Recipe_Tray_Meaurement D20.06 BOOL  ; Enable for Tray Measurement
Loaded_Recipe_Tray_Position D62 UINT
Loaded_Recipe_Tray_Settle_Time D56 UINT
Loaded_Recipe_Tray_Stop_Delay D53 UINT
Loaded_Recipe_Tray_height_measurement_enable D20.07 BOOL  ; Enables Height measurement of trays
Loaded_Recipe_Tray_measurement_Time D112 UINT  ; Time to measure tray
Loaded_Recipe_Upstream_Off_Delay D61 UINT
Loaded_Recipe_Upstream_On_Delay D60 UINT
Loaded_Recipe_VAC_Type D20.00 BOOL  ; Vac type - ON = Pressure, OFF = Time
Loaded_Recipe_Vacuum_Duration D37 UINT
Loaded_Recipe_Vacuum_Extra_Time D39 UINT
Loaded_Recipe_Vacuum_Pressure_SP D38 UINT
Loaded_Recipe_Vent_Bottom_Delay D44 UINT
Loaded_Recipe_Vent_Duration D45 UINT
Loaded_Recipe_Vent_Pressure_SP D46 UINT
Loaded_Recipe_Vent_Top_Delay D43 UINT
Loaded_Recipe_Vent_Type D20.02 BOOL  ; Vent type - ON = Pressure, OFF = Time
Loaded_Recipe_max_tray_size D116 UINT  ; maximum tray size
Loop1_AT_Delay T0270 TIMER  ; Delay to Start Loop1 Auto Tune
Loop1_CP_Feedback D20233 UINT
Loop1_D_Feedback D20237 UINT
Loop1_I_Feedback D20236 UINT
Loop1_P_Feedback D20235 UINT
Loop2_AT_Delay T0271 TIMER  ; Delay to Start Loop2 Auto Tune
Loop2_CP_Feedback D20243 UINT
Loop2_D_Feedback D20247 UINT
Loop2_I_Feedback D20246 UINT
Loop2_P_Feedback D20245 UINT
Loop3_AT_Delay T0272 TIMER  ; Delay to Start Loop3 Auto Tune
Loop3_CP_Feedback D20273 UINT
Loop3_D_Feedback D20277 UINT
Loop3_I_Feedback D20276 UINT
Loop3_P_Feedback D20275 UINT
Loop4_AT_Delay T0273 TIMER  ; Delay to Start Loop4 Auto Tune
Loop4_CP_Feedback D20283 UINT
Loop4_D_Feedback D20287 UINT
Loop4_I_Feedback D20286 UINT
Loop4_P_Feedback D20285 UINT
Loop5_AT_Delay T0274 TIMER  ; Delay to Start Loop5 Auto Tune
Loop5_CP_Feedback D21233 UINT
Loop5_D_Feedback D21237 UINT
Loop5_I_Feedback D21236 UINT
Loop5_P_Feedback D21235 UINT
Loop6_AT_Delay T0275 TIMER  ; Delay to Start Loop6 Auto Tune
Loop6_CP_Feedback D21243 UINT
Loop6_D_Feedback D21247 UINT
Loop6_I_Feedback D21246 UINT
Loop6_P_Feedback D21245 UINT
Low_Temp_Tol_CtoF offsetC_to_offsetF
Low_Temp_Tol_FtoC OffsetF_to_OffsetC
Low_Temp_delay T0141 TIMER  ; Delay for Low Temp Fault
Lower_Tool_Pressure 2007 UINT  ; Lower Tool pressure
Lower_Vac_Duration_Simultaneous_Timer T0207 TIMER  ; Used for simultaneous Mode
MAP_Mode W201.03 BOOL
MV_Lower_Limit_Heater1 D6007 UINT  ; Lower limit for MV if bit 12 of D5005 is on.
MV_Lower_Limit_Heater2 D6057 UINT  ; Lower limit for MV if bit 12 of D6005 is on.
MV_Lower_Limit_Heater3 D6107 UINT  ; Lower limit for MV if bit 12 of D6005 is on.
MV_Lower_Limit_Heater4 D6157 UINT  ; Lower limit for MV if bit 12 of D6005 is on.
MV_Lower_Limit_Heater5 D6207 UINT  ; Lower limit for MV if bit 12 of D6005 is on.
MV_Upper_Limit_Heater1 D6008 UINT  ; Upper limit for MV if bit 12 of D5005 is on.
MV_Upper_Limit_Heater2 D6058 UINT  ; Upper limit for MV if bit 12 of D6005 is on.
MV_Upper_Limit_Heater3 D6108 UINT  ; Upper limit for MV if bit 12 of D6005 is on.
MV_Upper_Limit_Heater4 D6158 UINT  ; Upper limit for MV if bit 12 of D6005 is on.
MV_Upper_Limit_Heater5 D6208 UINT  ; Upper limit for MV if bit 12 of D6005 is on.
Manual_Film_Single_Feed W200.06 BOOL  ; Manual button for film feed - 1 cycle
Manual_Film_Slow_Jog W200.07 BOOL  ; Manual button for film feed slow jog (hold button down)
Map_Seq_Step_Number D511 UINT  ; Contains the step number for the map sequence
Max_Temp_To_Run D1139 UINT  ; Maximum temperature allowed to run the machine
Measured_Tray_Time D600 UINT  ; Measured Tray Time
Measured_cycle_Time D2009.12 BOOL  ; Measured_cycle_Time
Measuremnt_alarm_latch W156.00 BOOL  ; Memory bit for measuremnt alarm
Memory_Card_Detected_Flag A343.15 BOOL  ; The memory card is inserted
Min_Dist_Calc_1 Minimum_Distance_Calc
Min_Temp_To_Run D1136 UINT  ; Minimum temperature to run the machine
Minimum_Calculated_Dist W400 DINT  ; Minimum distance setting
Missed_Tray_Timer T0110 TIMER  ; Missed tray timer
Move_parameters_start_film D2204.00 BOOL
No_Servo W202.14 BOOL  ; No servo on this machine
NotUsedTray6_AT_On_Flag 2129.03 BOOL  ; Loop6 Auto Tune ON
NotUsedTray6_ChangePIDConstants 2122.12 BOOL  ; Loop6 Turn Off PID constant flag
NotUsedTray6_Constants_Calculated 2129.10 BOOL  ; Loop6 PID Constants Calc flag
NotUsedTray6_FATALCONTROL_Error 2129.12 BOOL  ; Loop6 FATAL CONTROL Error
NotUsedTray6_Output_On 2129.04 BOOL  ; Loop6 Control Output ON
NotUsedTray6_PID_Save 2122.14 BOOL  ; Loop6 Save to EEPROM
NotUsedTray6_PV 2124 INT  ; Loop6 Process Value
NotUsedTray6_SENSOR_Error 2129.14 BOOL  ; Loop6 SENSOR error
NotUsedTray6_SETTING_Error 2129.09 BOOL  ; Loop6 SETTING Error
NotUsedTray6_SP 2121 INT  ; Loop 6 Setpoint
NotUsedTray6_Save_Complete 2129.15 BOOL  ; Loop6 Save to EEPROM complete
NotUsedTray6_Start_AT 2122.00 BOOL  ; Loop6 Start Auto Tune
NotUsedTray6_Stop 2122.04 BOOL  ; Loop6 Stop Controlling
NotUsedTray6_Stop_AT 2122.01 BOOL  ; Loop6 Stop Auto Tune
Not_Used_Loop_7_CP_Feedback D21273 UINT
Not_Used_Loop_7_D_Feedback D21277 UINT
Not_Used_Loop_7_I_Feedback D21276 UINT
Not_Used_Loop_7_P_Feedback D21275 UINT
Not_Used_Loop_8_CP_Feedback D21283 UINT
Not_Used_Loop_8_D_Feedback D21287 UINT
Not_Used_Loop_8_I_Feedback D21286 UINT
Not_Used_Loop_8_P_Feedback D21285 UINT
Not_Used_Tray7and8_Alarm_Mode D21201 CHANNEL
Not_Used_Tray_7_AT_On_Flag 2138.03 BOOL  ; Loop7 Auto Tune ON
Not_Used_Tray_7_ChangePIDConstants 2132.13 BOOL  ; Loop7 Turn Off PID constant flag
Not_Used_Tray_7_Constants_Calculated 2138.10 BOOL  ; Loop7 PID Constants Calc flag
Not_Used_Tray_7_ControlPeriod_SP D21253 UINT
Not_Used_Tray_7_Derivative D21257 UINT
Not_Used_Tray_7_FATALCONTROL_Error 2138.12 BOOL  ; Loop7 FATAL CONTROL Error
Not_Used_Tray_7_Integral_Time D21256 UINT
Not_Used_Tray_7_Output_On 2138.04 BOOL  ; Loop7 Control Output ON
Not_Used_Tray_7_PID_Save 2132.15 BOOL  ; Loop7 Save to EEPROM
Not_Used_Tray_7_PV 2133 INT  ; Loop7 Process Value
Not_Used_Tray_7_Proportional D21255 UINT
Not_Used_Tray_7_SENSOR_Error 2138.14 BOOL  ; Loop7 SENSOR error
Not_Used_Tray_7_SETTING_Error 2138.09 BOOL  ; Loop7 SETTING Error
Not_Used_Tray_7_SP 2130 INT  ; Loop 7 Setpoint
Not_Used_Tray_7_Save_Complete 2138.15 BOOL  ; Loop7 Save to EEPROM complete
Not_Used_Tray_7_Start_AT 2132.02 BOOL  ; Loop7 Start Auto Tune
Not_Used_Tray_7_Stop 2132.06 BOOL  ; Loop7 Stop Controlling
Not_Used_Tray_7_StopAT 2132.03 BOOL  ; Loop7 Stop Auto Tune
Not_Used_Tray_8_AT_On_Flag 2139.03 BOOL  ; Loop8 Auto Tune ON
Not_Used_Tray_8_ChangePIDConstants 2132.12 BOOL  ; Loop8 Turn Off PID constant flag
Not_Used_Tray_8_Constants_Calculated 2139.10 BOOL  ; Loop8 PID Constants Calc flag
Not_Used_Tray_8_ControlPeriod_SP D21263 UINT
Not_Used_Tray_8_Derivative D21267 UINT
Not_Used_Tray_8_FATALCONTROL_Error 2139.12 BOOL  ; Loop8 FATAL CONTROL Error
Not_Used_Tray_8_Integral_Time D21266 UINT
Not_Used_Tray_8_Output_On 2139.04 BOOL  ; Loop8 Control Output ON
Not_Used_Tray_8_PID_Save 2132.14 BOOL  ; Loop8 Save to EEPROM
Not_Used_Tray_8_PV 2134 INT  ; Loop8 Process Value
Not_Used_Tray_8_Proportional D21265 UINT
Not_Used_Tray_8_SENSOR_Error 2139.14 BOOL  ; Loop8 SENSOR error
Not_Used_Tray_8_SETTING_Error 2139.09 BOOL  ; Loop8 SETTING Error
Not_Used_Tray_8_SP 2131 INT  ; Loop 8 Setpoint
Not_Used_Tray_8_Save_Complete 2139.15 BOOL  ; Loop8 Save to EEPROM complete
Not_Used_Tray_8_Start_AT 2132.00 BOOL  ; Loop8 Start Auto Tune
Not_Used_Tray_8_Stop 2132.04 BOOL  ; Loop8 Stop Controlling
Not_Used_Tray_8_Stop_AT 2132.01 BOOL  ; Loop8 Stop Auto Tune
Num_Of_Trays_set_to_0 W151.05 BOOL  ; The number of trays has been set to 0
OPEN_Gripper_Auto D2011.02 BOOL  ; Open Gripper auto command
OPEN_Grippers_Delay T0231 TIMER  ; Delay Gripper auto open
One_shot_averaging_scaling D2034.02 BOOL  ; one shot for averaging
Outfeed_Conveyor_Run 3.15 BOOL  ; Outfeed conveyor run
Outfeed_Conveyor_Timer T0222 TIMER  ; Sets minimum time for outfeed conveyor to run
Outfeed_Estop_Fault W151.00 BOOL  ; Outfeed E-Stop Pressed
Outfeed_Estop_OK 0.10 BOOL  ; E-Stop circuit status
OverTemp_Delay T0142 TIMER  ; Delay for Over Temperature Fault
Overall_Compare_result D3266 UINT  ; If the current recipe completely matches the last loaded recipe, this value is Hex FFFF
PIDAT_Ouput_Heater1 D6041 UINT  ; Output word for PIDAT function - 0 - 8191 range (13 bits)
PIDAT_Ouput_Heater2 D6091 UINT  ; Output word for PIDAT function - 0 - 8191 range (13 bits)
PIDAT_Ouput_Heater3 D6141 UINT  ; Output word for PIDAT function - 0 - 8191 range (13 bits)
PIDAT_Ouput_Heater4 D6191 UINT  ; Output word for PIDAT function - 0 - 8191 range (13 bits)
PIDAT_Ouput_Heater5 D6241 UINT  ; Output word for PIDAT function - 0 - 8191 range (13 bits)
PIDAT_Settings1_Heater1 D6005 CHANNEL  ; Alpha, constant timing, MV designation, Forward / reverse
PIDAT_Settings1_Heater2 D6055 CHANNEL  ; Alpha, constant timing, MV designation, Forward / reverse
PIDAT_Settings1_Heater3 D6105 CHANNEL  ; Alpha, constant timing, MV designation, Forward / reverse
PIDAT_Settings1_Heater4 D6155 CHANNEL  ; Alpha, constant timing, MV designation, Forward / reverse
PIDAT_Settings1_Heater5 D6205 CHANNEL  ; Alpha, constant timing, MV designation, Forward / reverse
PIDAT_Settings2_Heater1 D6006 CHANNEL  ; Integral MV designation, MV Limit enable / disable, Input / output ranges
PIDAT_Settings2_Heater2 D6056 CHANNEL  ; Integral MV designation, MV Limit enable / disable, Input / output ranges
PIDAT_Settings2_Heater3 D6106 CHANNEL  ; Integral MV designation, MV Limit enable / disable, Input / output ranges
PIDAT_Settings2_Heater4 D6156 CHANNEL  ; Integral MV designation, MV Limit enable / disable, Input / output ranges
PIDAT_Settings2_Heater5 D6206 CHANNEL  ; Integral MV designation, MV Limit enable / disable, Input / output ranges
PIDAT_Settings3_Heater1 D6009 CHANNEL  ; Bits 0 - 11 is the calculated gain from the Autotune function
PIDAT_Settings3_Heater2 D6059 CHANNEL  ; Bits 0 - 11 is the calculated gain from the Autotune function
PIDAT_Settings3_Heater3 D6109 CHANNEL  ; Bits 0 - 11 is the calculated gain from the Autotune function
PIDAT_Settings3_Heater4 D6159 CHANNEL  ; Bits 0 - 11 is the calculated gain from the Autotune function
PIDAT_Settings3_Heater5 D6209 CHANNEL  ; Bits 0 - 11 is the calculated gain from the Autotune function
PIDAT_Work_Area_Word10_Heater1 D6020 CHANNEL  ; Work area for PIDAT function - DO NOT USE FOR ANYTHING ELSE.
PIDAT_Work_Area_Word10_Heater2 D6070 CHANNEL  ; Work area for PIDAT function - DO NOT USE FOR ANYTHING ELSE.
PIDAT_Work_Area_Word10_Heater3 D6120 CHANNEL  ; Work area for PIDAT function - DO NOT USE FOR ANYTHING ELSE.
PIDAT_Work_Area_Word10_Heater4 D6170 CHANNEL  ; Work area for PIDAT function - DO NOT USE FOR ANYTHING ELSE.
PIDAT_Work_Area_Word10_Heater5 D6220 CHANNEL  ; Work area for PIDAT function - DO NOT USE FOR ANYTHING ELSE.
PIDAT_Work_Area_Word11_Heater1 D6021 CHANNEL  ; Work area for PIDAT function - DO NOT USE FOR ANYTHING ELSE.
PIDAT_Work_Area_Word11_Heater2 D6071 CHANNEL  ; Work area for PIDAT function - DO NOT USE FOR ANYTHING ELSE.
PIDAT_Work_Area_Word11_Heater3 D6121 CHANNEL  ; Work area for PIDAT function - DO NOT USE FOR ANYTHING ELSE.
PIDAT_Work_Area_Word11_Heater4 D6171 CHANNEL  ; Work area for PIDAT function - DO NOT USE FOR ANYTHING ELSE.
PIDAT_Work_Area_Word11_Heater5 D6221 CHANNEL  ; Work area for PIDAT function - DO NOT USE FOR ANYTHING ELSE.
PIDAT_Work_Area_Word12_Heater1 D6022 CHANNEL  ; Work area for PIDAT function - DO NOT USE FOR ANYTHING ELSE.
PIDAT_Work_Area_Word12_Heater2 D6072 CHANNEL  ; Work area for PIDAT function - DO NOT USE FOR ANYTHING ELSE.
PIDAT_Work_Area_Word12_Heater3 D6122 CHANNEL  ; Work area for PIDAT function - DO NOT USE FOR ANYTHING ELSE.
PIDAT_Work_Area_Word12_Heater4 D6172 CHANNEL  ; Work area for PIDAT function - DO NOT USE FOR ANYTHING ELSE.
PIDAT_Work_Area_Word12_Heater5 D6222 CHANNEL  ; Work area for PIDAT function - DO NOT USE FOR ANYTHING ELSE.
PIDAT_Work_Area_Word13_Heater1 D6023 CHANNEL  ; Work area for PIDAT function - DO NOT USE FOR ANYTHING ELSE.
PIDAT_Work_Area_Word13_Heater2 D6073 CHANNEL  ; Work area for PIDAT function - DO NOT USE FOR ANYTHING ELSE.
PIDAT_Work_Area_Word13_Heater3 D6123 CHANNEL  ; Work area for PIDAT function - DO NOT USE FOR ANYTHING ELSE.
PIDAT_Work_Area_Word13_Heater4 D6173 CHANNEL  ; Work area for PIDAT function - DO NOT USE FOR ANYTHING ELSE.
PIDAT_Work_Area_Word13_Heater5 D6223 CHANNEL  ; Work area for PIDAT function - DO NOT USE FOR ANYTHING ELSE.
PIDAT_Work_Area_Word14_Heater1 D6024 CHANNEL  ; Work area for PIDAT function - DO NOT USE FOR ANYTHING ELSE.
PIDAT_Work_Area_Word14_Heater2 D6074 CHANNEL  ; Work area for PIDAT function - DO NOT USE FOR ANYTHING ELSE.
PIDAT_Work_Area_Word14_Heater3 D6124 CHANNEL  ; Work area for PIDAT function - DO NOT USE FOR ANYTHING ELSE.
PIDAT_Work_Area_Word14_Heater4 D6174 CHANNEL  ; Work area for PIDAT function - DO NOT USE FOR ANYTHING ELSE.
PIDAT_Work_Area_Word14_Heater5 D6224 CHANNEL  ; Work area for PIDAT function - DO NOT USE FOR ANYTHING ELSE.
PIDAT_Work_Area_Word15_Heater1 D6025 CHANNEL  ; Work area for PIDAT function - DO NOT USE FOR ANYTHING ELSE.
PIDAT_Work_Area_Word15_Heater2 D6075 CHANNEL  ; Work area for PIDAT function - DO NOT USE FOR ANYTHING ELSE.
PIDAT_Work_Area_Word15_Heater3 D6125 CHANNEL  ; Work area for PIDAT function - DO NOT USE FOR ANYTHING ELSE.
PIDAT_Work_Area_Word15_Heater4 D6175 CHANNEL  ; Work area for PIDAT function - DO NOT USE FOR ANYTHING ELSE.
PIDAT_Work_Area_Word15_Heater5 D6225 CHANNEL  ; Work area for PIDAT function - DO NOT USE FOR ANYTHING ELSE.
PIDAT_Work_Area_Word16_Heater1 D6026 CHANNEL  ; Work area for PIDAT function - DO NOT USE FOR ANYTHING ELSE.
PIDAT_Work_Area_Word16_Heater2 D6076 CHANNEL  ; Work area for PIDAT function - DO NOT USE FOR ANYTHING ELSE.
PIDAT_Work_Area_Word16_Heater3 D6126 CHANNEL  ; Work area for PIDAT function - DO NOT USE FOR ANYTHING ELSE.
PIDAT_Work_Area_Word16_Heater4 D6176 CHANNEL  ; Work area for PIDAT function - DO NOT USE FOR ANYTHING ELSE.
PIDAT_Work_Area_Word16_Heater5 D6226 CHANNEL  ; Work area for PIDAT function - DO NOT USE FOR ANYTHING ELSE.
PIDAT_Work_Area_Word17_Heater1 D6027 CHANNEL  ; Work area for PIDAT function - DO NOT USE FOR ANYTHING ELSE.
PIDAT_Work_Area_Word17_Heater2 D6077 CHANNEL  ; Work area for PIDAT function - DO NOT USE FOR ANYTHING ELSE.
PIDAT_Work_Area_Word17_Heater3 D6127 CHANNEL  ; Work area for PIDAT function - DO NOT USE FOR ANYTHING ELSE.
PIDAT_Work_Area_Word17_Heater4 D6177 CHANNEL  ; Work area for PIDAT function - DO NOT USE FOR ANYTHING ELSE.
PIDAT_Work_Area_Word17_Heater5 D6227 CHANNEL  ; Work area for PIDAT function - DO NOT USE FOR ANYTHING ELSE.
PIDAT_Work_Area_Word18_Heater1 D6028 CHANNEL  ; Work area for PIDAT function - DO NOT USE FOR ANYTHING ELSE.
PIDAT_Work_Area_Word18_Heater2 D6078 CHANNEL  ; Work area for PIDAT function - DO NOT USE FOR ANYTHING ELSE.
PIDAT_Work_Area_Word18_Heater3 D6128 CHANNEL  ; Work area for PIDAT function - DO NOT USE FOR ANYTHING ELSE.
PIDAT_Work_Area_Word18_Heater4 D6178 CHANNEL  ; Work area for PIDAT function - DO NOT USE FOR ANYTHING ELSE.
PIDAT_Work_Area_Word18_Heater5 D6228 CHANNEL  ; Work area for PIDAT function - DO NOT USE FOR ANYTHING ELSE.
PIDAT_Work_Area_Word19_Heater1 D6029 CHANNEL  ; Work area for PIDAT function - DO NOT USE FOR ANYTHING ELSE.
PIDAT_Work_Area_Word19_Heater2 D6079 CHANNEL  ; Work area for PIDAT function - DO NOT USE FOR ANYTHING ELSE.
PIDAT_Work_Area_Word19_Heater3 D6129 CHANNEL  ; Work area for PIDAT function - DO NOT USE FOR ANYTHING ELSE.
PIDAT_Work_Area_Word19_Heater4 D6179 CHANNEL  ; Work area for PIDAT function - DO NOT USE FOR ANYTHING ELSE.
PIDAT_Work_Area_Word19_Heater5 D6229 CHANNEL  ; Work area for PIDAT function - DO NOT USE FOR ANYTHING ELSE.
PIDAT_Work_Area_Word1_Heater1 D6011 CHANNEL  ; Work area for PIDAT function - DO NOT USE FOR ANYTHING ELSE.
PIDAT_Work_Area_Word1_Heater2 D6061 CHANNEL  ; Work area for PIDAT function - DO NOT USE FOR ANYTHING ELSE.
PIDAT_Work_Area_Word1_Heater3 D6111 CHANNEL  ; Work area for PIDAT function - DO NOT USE FOR ANYTHING ELSE.
PIDAT_Work_Area_Word1_Heater4 D6161 CHANNEL  ; Work area for PIDAT function - DO NOT USE FOR ANYTHING ELSE.
PIDAT_Work_Area_Word1_Heater5 D6211 CHANNEL  ; Work area for PIDAT function - DO NOT USE FOR ANYTHING ELSE.
PIDAT_Work_Area_Word20_Heater1 D6030 CHANNEL  ; Work area for PIDAT function - DO NOT USE FOR ANYTHING ELSE.
PIDAT_Work_Area_Word20_Heater2 D6080 CHANNEL  ; Work area for PIDAT function - DO NOT USE FOR ANYTHING ELSE.
PIDAT_Work_Area_Word20_Heater3 D6130 CHANNEL  ; Work area for PIDAT function - DO NOT USE FOR ANYTHING ELSE.
PIDAT_Work_Area_Word20_Heater4 D6180 CHANNEL  ; Work area for PIDAT function - DO NOT USE FOR ANYTHING ELSE.
PIDAT_Work_Area_Word20_Heater5 D6230 CHANNEL  ; Work area for PIDAT function - DO NOT USE FOR ANYTHING ELSE.
PIDAT_Work_Area_Word21_Heater1 D6031 CHANNEL  ; Work area for PIDAT function - DO NOT USE FOR ANYTHING ELSE.
PIDAT_Work_Area_Word21_Heater2 D6081 CHANNEL  ; Work area for PIDAT function - DO NOT USE FOR ANYTHING ELSE.
PIDAT_Work_Area_Word21_Heater3 D6131 CHANNEL  ; Work area for PIDAT function - DO NOT USE FOR ANYTHING ELSE.
PIDAT_Work_Area_Word21_Heater4 D6181 CHANNEL  ; Work area for PIDAT function - DO NOT USE FOR ANYTHING ELSE.
PIDAT_Work_Area_Word21_Heater5 D6231 CHANNEL  ; Work area for PIDAT function - DO NOT USE FOR ANYTHING ELSE.
PIDAT_Work_Area_Word22_Heater1 D6032 CHANNEL  ; Work area for PIDAT function - DO NOT USE FOR ANYTHING ELSE.
PIDAT_Work_Area_Word22_Heater2 D6082 CHANNEL  ; Work area for PIDAT function - DO NOT USE FOR ANYTHING ELSE.
PIDAT_Work_Area_Word22_Heater3 D6132 CHANNEL  ; Work area for PIDAT function - DO NOT USE FOR ANYTHING ELSE.
PIDAT_Work_Area_Word22_Heater4 D6182 CHANNEL  ; Work area for PIDAT function - DO NOT USE FOR ANYTHING ELSE.
PIDAT_Work_Area_Word22_Heater5 D6232 CHANNEL  ; Work area for PIDAT function - DO NOT USE FOR ANYTHING ELSE.
PIDAT_Work_Area_Word23_Heater1 D6033 CHANNEL  ; Work area for PIDAT function - DO NOT USE FOR ANYTHING ELSE.
PIDAT_Work_Area_Word23_Heater2 D6083 CHANNEL  ; Work area for PIDAT function - DO NOT USE FOR ANYTHING ELSE.
PIDAT_Work_Area_Word23_Heater3 D6133 CHANNEL  ; Work area for PIDAT function - DO NOT USE FOR ANYTHING ELSE.
PIDAT_Work_Area_Word23_Heater4 D6183 CHANNEL  ; Work area for PIDAT function - DO NOT USE FOR ANYTHING ELSE.
PIDAT_Work_Area_Word23_Heater5 D6233 CHANNEL  ; Work area for PIDAT function - DO NOT USE FOR ANYTHING ELSE.
PIDAT_Work_Area_Word24_Heater1 D6034 CHANNEL  ; Work area for PIDAT function - DO NOT USE FOR ANYTHING ELSE.
PIDAT_Work_Area_Word24_Heater2 D6084 CHANNEL  ; Work area for PIDAT function - DO NOT USE FOR ANYTHING ELSE.
PIDAT_Work_Area_Word24_Heater3 D6134 CHANNEL  ; Work area for PIDAT function - DO NOT USE FOR ANYTHING ELSE.
PIDAT_Work_Area_Word24_Heater4 D6184 CHANNEL  ; Work area for PIDAT function - DO NOT USE FOR ANYTHING ELSE.
PIDAT_Work_Area_Word24_Heater5 D6234 CHANNEL  ; Work area for PIDAT function - DO NOT USE FOR ANYTHING ELSE.
PIDAT_Work_Area_Word25_Heater1 D6035 CHANNEL  ; Work area for PIDAT function - DO NOT USE FOR ANYTHING ELSE.
PIDAT_Work_Area_Word25_Heater2 D6085 CHANNEL  ; Work area for PIDAT function - DO NOT USE FOR ANYTHING ELSE.
PIDAT_Work_Area_Word25_Heater3 D6135 CHANNEL  ; Work area for PIDAT function - DO NOT USE FOR ANYTHING ELSE.
PIDAT_Work_Area_Word25_Heater4 D6185 CHANNEL  ; Work area for PIDAT function - DO NOT USE FOR ANYTHING ELSE.
PIDAT_Work_Area_Word25_Heater5 D6235 CHANNEL  ; Work area for PIDAT function - DO NOT USE FOR ANYTHING ELSE.
PIDAT_Work_Area_Word26_Heater1 D6036 CHANNEL  ; Work area for PIDAT function - DO NOT USE FOR ANYTHING ELSE.
PIDAT_Work_Area_Word26_Heater2 D6086 CHANNEL  ; Work area for PIDAT function - DO NOT USE FOR ANYTHING ELSE.
PIDAT_Work_Area_Word26_Heater3 D6136 CHANNEL  ; Work area for PIDAT function - DO NOT USE FOR ANYTHING ELSE.
PIDAT_Work_Area_Word26_Heater4 D6186 CHANNEL  ; Work area for PIDAT function - DO NOT USE FOR ANYTHING ELSE.
PIDAT_Work_Area_Word26_Heater5 D6236 CHANNEL  ; Work area for PIDAT function - DO NOT USE FOR ANYTHING ELSE.
PIDAT_Work_Area_Word27_Heater1 D6037 CHANNEL  ; Work area for PIDAT function - DO NOT USE FOR ANYTHING ELSE.
PIDAT_Work_Area_Word27_Heater2 D6087 CHANNEL  ; Work area for PIDAT function - DO NOT USE FOR ANYTHING ELSE.
PIDAT_Work_Area_Word27_Heater3 D6137 CHANNEL  ; Work area for PIDAT function - DO NOT USE FOR ANYTHING ELSE.
PIDAT_Work_Area_Word27_Heater4 D6187 CHANNEL  ; Work area for PIDAT function - DO NOT USE FOR ANYTHING ELSE.
PIDAT_Work_Area_Word27_Heater5 D6237 CHANNEL  ; Work area for PIDAT function - DO NOT USE FOR ANYTHING ELSE.
PIDAT_Work_Area_Word28_Heater1 D6038 CHANNEL  ; Work area for PIDAT function - DO NOT USE FOR ANYTHING ELSE.
PIDAT_Work_Area_Word28_Heater2 D6088 CHANNEL  ; Work area for PIDAT function - DO NOT USE FOR ANYTHING ELSE.
PIDAT_Work_Area_Word28_Heater3 D6138 CHANNEL  ; Work area for PIDAT function - DO NOT USE FOR ANYTHING ELSE.
PIDAT_Work_Area_Word28_Heater4 D6188 CHANNEL  ; Work area for PIDAT function - DO NOT USE FOR ANYTHING ELSE.
PIDAT_Work_Area_Word28_Heater5 D6238 CHANNEL  ; Work area for PIDAT function - DO NOT USE FOR ANYTHING ELSE.
PIDAT_Work_Area_Word29_Heater1 D6039 CHANNEL  ; Work area for PIDAT function - DO NOT USE FOR ANYTHING ELSE.
PIDAT_Work_Area_Word29_Heater2 D6089 CHANNEL  ; Work area for PIDAT function - DO NOT USE FOR ANYTHING ELSE.
PIDAT_Work_Area_Word29_Heater3 D6139 CHANNEL  ; Work area for PIDAT function - DO NOT USE FOR ANYTHING ELSE.
PIDAT_Work_Area_Word29_Heater4 D6189 CHANNEL  ; Work area for PIDAT function - DO NOT USE FOR ANYTHING ELSE.
PIDAT_Work_Area_Word29_Heater5 D6239 CHANNEL  ; Work area for PIDAT function - DO NOT USE FOR ANYTHING ELSE.
PIDAT_Work_Area_Word2_Heater1 D6012 CHANNEL  ; Work area for PIDAT function - DO NOT USE FOR ANYTHING ELSE.
PIDAT_Work_Area_Word2_Heater2 D6062 CHANNEL  ; Work area for PIDAT function - DO NOT USE FOR ANYTHING ELSE.
PIDAT_Work_Area_Word2_Heater3 D6112 CHANNEL  ; Work area for PIDAT function - DO NOT USE FOR ANYTHING ELSE.
PIDAT_Work_Area_Word2_Heater4 D6162 CHANNEL  ; Work area for PIDAT function - DO NOT USE FOR ANYTHING ELSE.
PIDAT_Work_Area_Word2_Heater5 D6212 CHANNEL  ; Work area for PIDAT function - DO NOT USE FOR ANYTHING ELSE.
PIDAT_Work_Area_Word30_Heater1 D6040 CHANNEL  ; Work area for PIDAT function - DO NOT USE FOR ANYTHING ELSE.
PIDAT_Work_Area_Word30_Heater2 D6090 CHANNEL  ; Work area for PIDAT function - DO NOT USE FOR ANYTHING ELSE.
PIDAT_Work_Area_Word30_Heater3 D6140 CHANNEL  ; Work area for PIDAT function - DO NOT USE FOR ANYTHING ELSE.
PIDAT_Work_Area_Word30_Heater4 D6190 CHANNEL  ; Work area for PIDAT function - DO NOT USE FOR ANYTHING ELSE.
PIDAT_Work_Area_Word30_Heater5 D6240 CHANNEL  ; Work area for PIDAT function - DO NOT USE FOR ANYTHING ELSE.
PIDAT_Work_Area_Word3_Heater1 D6013 CHANNEL  ; Work area for PIDAT function - DO NOT USE FOR ANYTHING ELSE.
PIDAT_Work_Area_Word3_Heater2 D6063 CHANNEL  ; Work area for PIDAT function - DO NOT USE FOR ANYTHING ELSE.
PIDAT_Work_Area_Word3_Heater3 D6113 CHANNEL  ; Work area for PIDAT function - DO NOT USE FOR ANYTHING ELSE.
PIDAT_Work_Area_Word3_Heater4 D6163 CHANNEL  ; Work area for PIDAT function - DO NOT USE FOR ANYTHING ELSE.
PIDAT_Work_Area_Word3_Heater5 D6213 CHANNEL  ; Work area for PIDAT function - DO NOT USE FOR ANYTHING ELSE.
PIDAT_Work_Area_Word4_Heater1 D6014 CHANNEL  ; Work area for PIDAT function - DO NOT USE FOR ANYTHING ELSE.
PIDAT_Work_Area_Word4_Heater2 D6064 CHANNEL  ; Work area for PIDAT function - DO NOT USE FOR ANYTHING ELSE.
PIDAT_Work_Area_Word4_Heater3 D6114 CHANNEL  ; Work area for PIDAT function - DO NOT USE FOR ANYTHING ELSE.
PIDAT_Work_Area_Word4_Heater4 D6164 CHANNEL  ; Work area for PIDAT function - DO NOT USE FOR ANYTHING ELSE.
PIDAT_Work_Area_Word4_Heater5 D6214 CHANNEL  ; Work area for PIDAT function - DO NOT USE FOR ANYTHING ELSE.
PIDAT_Work_Area_Word5_Heater1 D6015 CHANNEL  ; Work area for PIDAT function - DO NOT USE FOR ANYTHING ELSE.
PIDAT_Work_Area_Word5_Heater2 D6065 CHANNEL  ; Work area for PIDAT function - DO NOT USE FOR ANYTHING ELSE.
PIDAT_Work_Area_Word5_Heater3 D6115 CHANNEL  ; Work area for PIDAT function - DO NOT USE FOR ANYTHING ELSE.
PIDAT_Work_Area_Word5_Heater4 D6165 CHANNEL  ; Work area for PIDAT function - DO NOT USE FOR ANYTHING ELSE.
PIDAT_Work_Area_Word5_Heater5 D6215 CHANNEL  ; Work area for PIDAT function - DO NOT USE FOR ANYTHING ELSE.
PIDAT_Work_Area_Word6_Heater1 D6016 CHANNEL  ; Work area for PIDAT function - DO NOT USE FOR ANYTHING ELSE.
PIDAT_Work_Area_Word6_Heater2 D6066 CHANNEL  ; Work area for PIDAT function - DO NOT USE FOR ANYTHING ELSE.
PIDAT_Work_Area_Word6_Heater3 D6116 CHANNEL  ; Work area for PIDAT function - DO NOT USE FOR ANYTHING ELSE.
PIDAT_Work_Area_Word6_Heater4 D6166 CHANNEL  ; Work area for PIDAT function - DO NOT USE FOR ANYTHING ELSE.
PIDAT_Work_Area_Word6_Heater5 D6216 CHANNEL  ; Work area for PIDAT function - DO NOT USE FOR ANYTHING ELSE.
PIDAT_Work_Area_Word7_Heater1 D6017 CHANNEL  ; Work area for PIDAT function - DO NOT USE FOR ANYTHING ELSE.
PIDAT_Work_Area_Word7_Heater2 D6067 CHANNEL  ; Work area for PIDAT function - DO NOT USE FOR ANYTHING ELSE.
PIDAT_Work_Area_Word7_Heater3 D6117 CHANNEL  ; Work area for PIDAT function - DO NOT USE FOR ANYTHING ELSE.
PIDAT_Work_Area_Word7_Heater4 D6167 CHANNEL  ; Work area for PIDAT function - DO NOT USE FOR ANYTHING ELSE.
PIDAT_Work_Area_Word7_Heater5 D6217 CHANNEL  ; Work area for PIDAT function - DO NOT USE FOR ANYTHING ELSE.
PIDAT_Work_Area_Word8_Heater1 D6018 CHANNEL  ; Work area for PIDAT function - DO NOT USE FOR ANYTHING ELSE.
PIDAT_Work_Area_Word8_Heater2 D6068 CHANNEL  ; Work area for PIDAT function - DO NOT USE FOR ANYTHING ELSE.
PIDAT_Work_Area_Word8_Heater3 D6118 CHANNEL  ; Work area for PIDAT function - DO NOT USE FOR ANYTHING ELSE.
PIDAT_Work_Area_Word8_Heater4 D6168 CHANNEL  ; Work area for PIDAT function - DO NOT USE FOR ANYTHING ELSE.
PIDAT_Work_Area_Word8_Heater5 D6218 CHANNEL  ; Work area for PIDAT function - DO NOT USE FOR ANYTHING ELSE.
PIDAT_Work_Area_Word9_Heater1 D6019 CHANNEL  ; Work area for PIDAT function - DO NOT USE FOR ANYTHING ELSE.
PIDAT_Work_Area_Word9_Heater2 D6069 CHANNEL  ; Work area for PIDAT function - DO NOT USE FOR ANYTHING ELSE.
PIDAT_Work_Area_Word9_Heater3 D6119 CHANNEL  ; Work area for PIDAT function - DO NOT USE FOR ANYTHING ELSE.
PIDAT_Work_Area_Word9_Heater4 D6169 CHANNEL  ; Work area for PIDAT function - DO NOT USE FOR ANYTHING ELSE.
PIDAT_Work_Area_Word9_Heater5 D6219 CHANNEL  ; Work area for PIDAT function - DO NOT USE FOR ANYTHING ELSE.
PID_Global_AT T0236 TIMER  ; Delay to Start Global Auto Tune
PID_Mode H500.00 BOOL  ; Default PID =ON, Custom =OFF
PID_Mode_Change T0235 TIMER  ; Delay to change PID Control mode
PID_PROM_Save T0237 TIMER  ; Delay to Save to EEPROM
Pockets_in_tool_minus_one D245 UINT  ; Trays in tool minus 1
PositionFeedback_div_10 D880 DINT
Pressure_Transducer_disconnected 2009.06 BOOL  ; Input signal disconnected
Print_Delay_Timer T1101 TIMER  ; Print delay to Printer
Print_output_timer T1100 TIMER  ; Time to keep print signal on
Printed_Film_parameter_changed D2204.03 BOOL  ; Printed film parameter has changed
Printer_Enable 4.14 BOOL  ; Bell-Mark Printer Enable
Printer_Fault W153.15 BOOL  ; Bell-Mark Printer Fault
Printer_Faulted 1.15 BOOL  ; Bell-Mark Printer
Printer_Installed D2100.00 BOOL  ; The Bell-Mark Printer is installed on the machine
Printer_Print 4.15 BOOL  ; Bell-Mark Printer Print
Printer_Ready 1.14 BOOL  ; Bell-Mark Printer
Printer_not_Ready_Fault W153.14 BOOL  ; Bell-Mark Printer not ready
Q3_Heat_Contactor 2.00 BOOL  ; Q3 Tool Heat Contactor On output
REG_STOP_DECEL H35 UINT
REG_STOP_TARGET_FREQ H36 DINT  ; H36/H37
RET_ACC D888 DINT
RET_ACC_4ms D1108 UINT
RET_DEC D890 DINT
RET_DEC_4ms D1112 UINT
RET_Movement_Calcs Vel_ACC_DEC_Scale
RET_VEL D892 DINT
RTD_Dummy W500.00 BOOL  ; RTD Detected Dummy
Rear_Gripper_Closed_Prox 1.06 BOOL  ; IN650-850 Rear Gripper Closed Prox
Rear_Gripper_Open_Prox 1.05 BOOL  ; IN650-850 Rear Gripper Open Prox
Recipe_Compare_Match_0_15 D3250 WORD  ; Result of MCMP Instruction - 16 Match Conditions
Recipe_Compare_Match_112_127 D3257 WORD  ; Result of MCMP Instruction - 16 Match Conditions
Recipe_Compare_Match_128_143 D3258 WORD  ; Result of MCMP Instruction - 16 Match Conditions
Recipe_Compare_Match_144_159 D3259 WORD  ; Result of MCMP Instruction - 16 Match Conditions
Recipe_Compare_Match_160_175 D3260 WORD  ; Result of MCMP Instruction - 16 Match Conditions
Recipe_Compare_Match_16_31 D3251 WORD  ; Result of MCMP Instruction - 16 Match Conditions
Recipe_Compare_Match_176_191 D3261 WORD  ; Result of MCMP Instruction - 16 Match Conditions
Recipe_Compare_Match_192_207 D3262 WORD  ; Result of MCMP Instruction - 16 Match Conditions
Recipe_Compare_Match_208_223 D3263 WORD  ; Result of MCMP Instruction - 16 Match Conditions
Recipe_Compare_Match_224_239 D3264 WORD  ; Result of MCMP Instruction - 16 Match Conditions
Recipe_Compare_Match_234_249 D3265 WORD  ; Result of MCMP Instruction - 16 Match Conditions - Overlap with previouis to end right at 249
Recipe_Compare_Match_32_47 D3252 WORD  ; Result of MCMP Instruction - 16 Match Conditions
Recipe_Compare_Match_48_63 D3253 WORD  ; Result of MCMP Instruction - 16 Match Conditions
Recipe_Compare_Match_64_79 D3254 WORD  ; Result of MCMP Instruction - 16 Match Conditions
Recipe_Compare_Match_80_95 D3255 WORD  ; Result of MCMP Instruction - 16 Match Conditions
Recipe_Compare_Match_96_111 D3256 WORD  ; Result of MCMP Instruction - 16 Match Conditions
Recipe_End_Pointer E30003 UINT  ; End pointer for use with BSET command
Recipe_Filename D1400 STRING[74]  ; Filename for recipe file name saved to Compact flash in CSV format
Recipe_List_Pointer E30001 UINT  ; Creates a list of 10 consecutive recipe names
Recipe_Name_Display_Pointer D506 UINT
Recipe_Number_Selected D500 UINT  ; The recipe number selected on the screen.
Recipe_Number_for_Loop E30002 UINT  ; Used to set the recipe number in the recipe tables
Recipe_Pointer E30000 UINT  ; Points to the first word of the selected recipe in the recipe memory area (E0 - E24999)
Recipe_Pointer_Calc D504 DINT  ; Points at the first word in the recipe storage area (E0 - E24999) for the selected recipe.
Recover_After_Break W203.06 BOOL
Recover_Count_Setting D961 UINT  ; HMI Setting
Recover_Feed W203.07 BOOL
Recover_count D962 UINT
Registration_Arming_Count D1117 UINT
Registration_Count D1118 UINT
Registration_Film_Feed_Fault W151.15 BOOL  ; Incorrect mark count or film didn't stop
Registration_Film_Feeding W200.13 BOOL  ; Film Feeding
Registration_Position_Fault W150.12 BOOL  ; Registration position incorrect at end of feed
Registration_Sensor 2960.00 BOOL  ; Input 0 on the MD card.
Reset_Servo_Timer T0201 TIMER  ; Timer for resetting servo
Reset_TPM D966.01 BOOL
Resettable_Cycle_Count D896 UDINT  ; Can be reset by operator
Return_Gripper_Tool_Change W203.04 BOOL  ; Return the Gripper to tool change position.
Reverse_Yank W200.11 BOOL  ; Reverse Yank
Reverse_Yank_Timer T0200 TIMER  ; Pause between reverse yank and moving forward
Rewind_Dancer_Up_Prox 0.00 BOOL  ; Proximity sw input
Rewind_Timout_WD_Fault W150.11 BOOL  ; Watchdog Timer Fault
Rewind_Timout_WD_Timer T0140 TIMER  ; Watchdog Timer
Run_latch W200.00 BOOL  ; Machine Run Latch
SP_HB1 D2005 CHANNEL  ; Heater burnout current 1
SP_HB2 D2006 CHANNEL  ; Heater burnout current 2
SP_HB3 D2007 CHANNEL  ; Heater burnout current 3
SP_HB4 D2008 CHANNEL  ; Heater burnout current 4
SSR1_Seal_Bar_1_Heat 2.01 BOOL  ; Seal Bar 1 Heat On output
SSR2_Seal_Bar_2_Heat 2.02 BOOL  ; Seal Bar 2 Heat On output
SSR3_Seal_Bar_3_Heat 4.00 BOOL  ; SSR3 Seal Bar 3 Heat output
SSR4_Seal_Bar_4_Heat 4.01 BOOL  ; SSR4 Seal Bar Heat 4 output
SSR5_Seal_Bar_5_Heat 4.02 BOOL  ; SSR 5 Seal Bar Heat output 5
SSR6_Rewind_Mtr_Starter 2.08 BOOL  ; SSR6 Rewind Motor Run output
Safeties_Clear W0.01 BOOL  ; All Machine guards, E-Stops OK
SafetyPopUp_FrontDoor W510.03 BOOL  ; Front door Safety
SafetyPopUp_InfeedEStop W510.01 BOOL  ; Pop_Up_estop_back
SafetyPopUp_InfeedGuard W510.04 BOOL  ; Pop_Up_Infeed_Gaurd
SafetyPopUp_OutFeedEStop W510.02 BOOL  ; Pop_Up_estop_front
SafetyPopUp_RearDoor W510.05 BOOL  ; Back door safety
Safety_Authority W0.00 BOOL  ; All Estops and doors OK - Internal Latched Status
Saved_Recipe_Val_FilmFeedACC D2201 UINT
Saved_Recipe_Val_FilmFeedDEC D2202 UINT
Saved_Recipe_Val_FilmFeedVel D2200 UINT
Scale_Analog_Out Conv_Scale_analog_with_Int_range
Scaled_result D2070 UINT
Seal_Bar_Pulse_Timer T0127 TIMER  ; Seal bar retract pulse timer
Seal_Bar_retract_delay T0216 TIMER  ; Retract delay after clamping
Seal_Delay_Timer T0122 TIMER  ; Seal_Delay_Timer
Seal_Duration_Timer T0123 TIMER  ; Seal Duration Timer
Seal_Recharge_Delay T0227 TIMER  ; Delay to recharge Seal valve
Seal_Recharge_Pulse T0228 TIMER  ; Pulse to recharge Seal valve
Seal_recharge D2009.11 BOOL  ; Seal Air charge
Selected_Pointer_Calc1 D513 UINT  ; Pointer calculation intermediate step
Selected_Pointer_Calc2 D514 DINT  ; Pointer calculation intermediate step 2
Selected_Recipe_Advance_Accel D322 UINT
Selected_Recipe_Advance_Decel D323 UINT
Selected_Recipe_Advance_Time D320 UINT
Selected_Recipe_Advance_Velocity D321 UINT
Selected_Recipe_Bottom_Vacuum_Delay D287 UINT
Selected_Recipe_Cycle_Type D280 UINT  ; Cycle type selection (Flat, Map, Simultaneous, VSP)
Selected_Recipe_Dancing_Stop D309 UINT
Selected_Recipe_Feed_Delay_After_Adv D303 UINT
Selected_Recipe_Film_Feed_Accel D327 UINT
Selected_Recipe_Film_Feed_Decel D328 UINT
Selected_Recipe_Film_Feed_Velocity D326 UINT
Selected_Recipe_Film_Jog_Accel D331 UINT
Selected_Recipe_Film_Jog_Decel D332 UINT
Selected_Recipe_Film_Jog_Velocity D330 UINT
Selected_Recipe_Film_Length D282 UINT  ; Film length to feed
Selected_Recipe_Gas_Delay D291 UINT
Selected_Recipe_Gas_Duration D292 UINT
Selected_Recipe_Gas_Pressure_SP D293 UINT
Selected_Recipe_Gas_Type D270.01 BOOL  ; Gas type - ON = Pressure, OFF = Time
Selected_Recipe_Grip_Open_Delay D318 UINT
Selected_Recipe_Gripper_ADV_Delay D308 UINT
Selected_Recipe_Gripper_Close_Delay D301 UINT
Selected_Recipe_Index D507 UINT  ; Selected recipe name on Recipe Screen
Selected_Recipe_Infeed_Gate_Eye_Debounce D306 UINT
Selected_Recipe_Infeed_speed D285 UINT  ; Infeed speed setting
Selected_Recipe_Job_Number_Display D1219 UINT  ; Recipe number of displayed recipe
Selected_Recipe_Job_Number_Display_Plus_1 D1239 UINT  ; Recipe number of displayed recipe
Selected_Recipe_Job_Number_Display_Plus_2 D1259 UINT  ; Recipe number of displayed recipe
Selected_Recipe_Job_Number_Display_Plus_3 D1279 UINT  ; Recipe number of displayed recipe
Selected_Recipe_Job_Number_Display_Plus_4 D1299 UINT  ; Recipe number of displayed recipe
Selected_Recipe_Job_Number_Display_Plus_5 D1319 UINT  ; Recipe number of displayed recipe
Selected_Recipe_Job_Number_Display_Plus_6 D1339 UINT  ; Recipe number of displayed recipe
Selected_Recipe_Job_Number_Display_Plus_7 D1359 UINT  ; Recipe number of displayed recipe
Selected_Recipe_Job_Number_Display_Plus_8 D1379 UINT  ; Recipe number of displayed recipe
Selected_Recipe_Job_Number_Display_Plus_9 D1399 UINT  ; Recipe number of displayed recipe
Selected_Recipe_Lift_Decel D324 UINT
Selected_Recipe_Lost_Tray_Reset_Delay D305 UINT
Selected_Recipe_Lower_Decel D325 UINT
Selected_Recipe_Motion_Setting_from_Time D270.05 BOOL  ; Chooses time setting or vel, accel and decel settings
Selected_Recipe_Name D250 STRING[38]  ; Job name for Recipe 0
Selected_Recipe_Name_Display D1200 STRING[38]  ; Selected recipe name for display in a list.
Selected_Recipe_Name_Display_plus_1 D1220 STRING[38]  ; Selected recipe name for display in a list.  Selected + 1
Selected_Recipe_Name_Display_plus_2 D1240 STRING[38]  ; Selected recipe name for display in a list.  Selected + 2
Selected_Recipe_Name_Display_plus_3 D1260 STRING[38]  ; Selected recipe name for display in a list.  Selected + 3
Selected_Recipe_Name_Display_plus_4 D1280 STRING[38]  ; Selected recipe name for display in a list.  Selected + 4
Selected_Recipe_Name_Display_plus_5 D1300 STRING[38]  ; Selected recipe name for display in a list.  Selected + 5
Selected_Recipe_Name_Display_plus_6 D1320 STRING[38]  ; Selected recipe name for display in a list.  Selected + 6
Selected_Recipe_Name_Display_plus_7 D1340 STRING[38]  ; Selected recipe name for display in a list.  Selected + 7
Selected_Recipe_Name_Display_plus_8 D1360 STRING[38]  ; Selected recipe name for display in a list.  Selected + 8
Selected_Recipe_Name_Display_plus_9 D1380 STRING[38]  ; Selected recipe name for display in a list.  Selected + 9
Selected_Recipe_Number D269 UINT  ; Recipe Number (0 - 99)
Selected_Recipe_Number_of_Trays D310 UINT
Selected_Recipe_REV_Yank D270.03 BOOL  ; On if reverse yank enabled for film
Selected_Recipe_Recipe_Number D279 UINT  ; Recipe Number
Selected_Recipe_Reg_Offset D284 UINT  ; Registration Offset
